(* CODESYS project KotelnayLesnay.project
   Title: KotelnayLesnay
   Author: User
   Version: 0.0.0.178

Project tree, tasks and I/O mapping:
  MyController : TM241CE40T/U, Schneider Electric, order no. TM241CE40T/U, version 4.0.6.18
    application Application
      libraries: Toolbox_Advance, 1.0.1.0 (Schneider Electric); Toolbox, 2.2.0.0 (Schneider Electric); SysTimeRtc, 3.5.1.0 (System)
      task MAST (cyclic, interval 20 ms, priority 15, watchdog 100 ms x 1) calls INPUT, AnalogSensers, PidMeteoVlv, PidGvs, ManualMode, year_month_day, DQ
      global variables GVL
      program INPUT [ST]
      program DQ [ST]
      program ManualMode [LD]
      program AnalogSensers [FBD]
      global variables GVL_RETAIN
      program PidMeteoVlv [FBD]
      function block OutputLimit [ST]
      program year_month_day [CFC]
      function block SendData [CFC]
      function CRC16 [ST]
      function block CRC_16 [ST]
      function block array_to_float [ST]
      data type word_real
      program PidGvs [FBD]
      function block InitializationTmpGrafik [ST]
    A1DI : Digital Inputs, Schneider Electric, version 4.0.6.18
        input  idwDI_IDW0 : DWORD  // IDW0
        input  X0 : BOOL  // IDW0.I0
        input  X1 : BOOL  // IDW0.I1
        input  X2 : BOOL  // IDW0.I2
        input  X3 : BOOL  // IDW0.I3
        input  X4 : BOOL  // IDW0.I4
        input  X5 : BOOL  // IDW0.I5
        input  X6 : BOOL  // IDW0.I6
        input  X7 : BOOL  // IDW0.I7
        input  X8 : BOOL  // IDW0.I8
        input  X9 : BOOL  // IDW0.I9
        input  X10 : BOOL  // IDW0.I10
        input  X11 : BOOL  // IDW0.I11
        input  X12 : BOOL  // IDW0.I12
        input  X13 : BOOL  // IDW0.I13
        input  X14 : BOOL  // IDW0.I14
        input  X15 : BOOL  // IDW0.I15
        input  X16 : BOOL  // IDW0.I16
        input  X17 : BOOL  // IDW0.I17
        input  X18 : BOOL  // IDW0.I18
        input  X19 : BOOL  // IDW0.I19
        input  X20 : BOOL  // IDW0.I20
        input  X21 : BOOL  // IDW0.I21
        input  X22 : BOOL  // IDW0.I22
        input  X23 : BOOL  // IDW0.I23
        input  ibDI_IB1 : BYTE  // IB1
    A1DQ : Digital Outputs, Schneider Electric, version 4.0.6.18
        output Y0 : BOOL  // QW0.Q0
        output Y1 : BOOL  // QW0.Q1
        output Y2 : BOOL  // QW0.Q2
        output Y3 : BOOL  // QW0.Q3
        output Y4 : BOOL  // QW0.Q4
        output Y5 : BOOL  // QW0.Q5
        output Y6 : BOOL  // QW0.Q6
        output Y7 : BOOL  // QW0.Q7
        output Y8 : BOOL  // QW0.Q8
        output Y9 : BOOL  // QW0.Q9
        output Y10 : BOOL  // QW0.Q10
        output Y11 : BOOL  // QW0.Q11
        output Y12 : BOOL  // QW0.Q12
        output Y13 : BOOL  // QW0.Q13
        output Y14 : BOOL  // QW0.Q14
        output Y15 : BOOL  // QW0.Q15
        output qbDQ_QB1 : BYTE  // QB1
        unmapped channels: QW0
    Counters : Counters, Schneider Electric, version 4.0.6.18
    Pulse_Generators : Pulse Generators, Schneider Electric, version 4.0.6.18
    Cartridge_1 : Cartridge, Schneider Electric, version 4.0.6.18
    Cartridge_2 : Cartridge, Schneider Electric, version 4.0.6.18
    IO_Bus : IO bus - TM3, Schneider Electric, version 4.0.6.18
      A12DI : TM3DI32K, Schneider Electric, order no. TM3DI32K, version 1.0.1.3
          input  idwModule_2_ID0 : DWORD  // ID0
          input  _1X0 : BOOL  // ID0.I0
          input  _1X1 : BOOL  // ID0.I1
          input  _1X2 : BOOL  // ID0.I2
          input  _1X3 : BOOL  // ID0.I3
          input  _1X4 : BOOL  // ID0.I4
          input  _1X5 : BOOL  // ID0.I5
          input  _1X6 : BOOL  // ID0.I6
          input  _1X7 : BOOL  // ID0.I7
          input  _1X8 : BOOL  // ID0.I8
          input  _1X9 : BOOL  // ID0.I9
          input  _1X10 : BOOL  // ID0.I10
          input  _1X11 : BOOL  // ID0.I11
          input  _1X12 : BOOL  // ID0.I12
          input  _1X13 : BOOL  // ID0.I13
          input  _1X14 : BOOL  // ID0.I14
          input  _1X15 : BOOL  // ID0.I15
          input  _1X16 : BOOL  // ID0.I16
          input  _1X17 : BOOL  // ID0.I17
          input  _1X18 : BOOL  // ID0.I18
          input  _1X19 : BOOL  // ID0.I19
          input  _1X24 : BOOL  // ID0.I24
          input  _1X25 : BOOL  // ID0.I25
          input  _1X23 : BOOL  // ID0.I27
          input  _1X20 : BOOL  // ID0.I28
          input  _1X21 : BOOL  // ID0.I29
          input  _1X22 : BOOL  // ID0.I30
      A13AI : TM3AI8/G, Schneider Electric, order no. TM3AI8/G, version 1.0.0.17
          settings: KPI Configuration.KPI Configuration[0] = 35; KPI Configuration.KPI Configuration[1] = 35; KPI Configuration.KPI Configuration[2] = 35; KPI Configuration.KPI Configuration[3] = 35; KPI Configuration.KPI Configuration[4] = 35; KPI Configuration.KPI Configuration[8] = 160; KPI Configuration.KPI Configuration[9] = 15; KPI Configuration.KPI Configuration[10] = 160; KPI Configuration.KPI Configuration[11] = 15; KPI Configuration.KPI Configuration[12] = 160; KPI Configuration.KPI Configuration[13] = 15; KPI Configuration.KPI Configuration[14] = 160; KPI Configuration.KPI Configuration[15] = 15; KPI Configuration.KPI Configuration[16] = 160; KPI Configuration.KPI Configuration[17] = 15; KPI Configuration.KPI Configuration[24] = 32; KPI Configuration.KPI Configuration[25] = 78; KPI Configuration.KPI Configuration[26] = 32; KPI Configuration.KPI Configuration[27] = 78; KPI Configuration.KPI Configuration[28] = 32; KPI Configuration.KPI Configuration[29] = 78; KPI Configuration.KPI Configuration[30] = 32; KPI Configuration.KPI Configuration[31] = 78; KPI Configuration.KPI Configuration[32] = 32; KPI Configuration.KPI Configuration[33] = 78; KPI Configuration.KPI Configuration[40] = 10; KPI Configuration.KPI Configuration[42] = 10; KPI Configuration.KPI Configuration[44] = 10; KPI Configuration.KPI Configuration[46] = 10; KPI Configuration.KPI Configuration[48] = 10
          input  PT3 : INT  // IW0
          input  PT4 : INT  // IW1
          input  PT6 : INT  // IW2
          input  PT5 : INT  // IW3
          input  PT8 : INT  // IW4
          input  PT10 : INT  // IW5
          input  iiModule_3_IW6 : INT  // IW6
          input  iiModule_3_IW7 : INT  // IW7
          input  ibModule_3_IBStatusIW0 : BYTE  // IBStatusIW0
          input  ibModule_3_IBStatusIW1 : BYTE  // IBStatusIW1
          input  ibModule_3_IBStatusIW2 : BYTE  // IBStatusIW2
          input  ibModule_3_IBStatusIW3 : BYTE  // IBStatusIW3
          input  ibModule_3_IBStatusIW4 : BYTE  // IBStatusIW4
          input  ibModule_3_IBStatusIW5 : BYTE  // IBStatusIW5
          input  ibModule_3_IBStatusIW6 : BYTE  // IBStatusIW6
          input  ibModule_3_IBStatusIW7 : BYTE  // IBStatusIW7
      A14AI : TM3TI4/G, Schneider Electric, order no. TM3TI4/G, version 1.0.1.5
          settings: KPI Configuration.KPI Configuration[0] = 77; KPI Configuration.KPI Configuration[1] = 77; KPI Configuration.KPI Configuration[2] = 77; KPI Configuration.KPI Configuration[3] = 77; KPI Configuration.KPI Configuration[4] = 48; KPI Configuration.KPI Configuration[5] = 248; KPI Configuration.KPI Configuration[6] = 48; KPI Configuration.KPI Configuration[7] = 248; KPI Configuration.KPI Configuration[8] = 48; KPI Configuration.KPI Configuration[9] = 248; KPI Configuration.KPI Configuration[10] = 48; KPI Configuration.KPI Configuration[11] = 248; KPI Configuration.KPI Configuration[12] = 52; KPI Configuration.KPI Configuration[13] = 33; KPI Configuration.KPI Configuration[14] = 52; KPI Configuration.KPI Configuration[15] = 33; KPI Configuration.KPI Configuration[16] = 52; KPI Configuration.KPI Configuration[17] = 33; KPI Configuration.KPI Configuration[18] = 52; KPI Configuration.KPI Configuration[19] = 33
          input  TE1 : INT  // IW0
          input  TE2 : INT  // IW1
          input  TE3 : INT  // IW2
          input  TE4 : INT  // IW3
          input  ibModule_4_IBStatusIW0 : BYTE  // IBStatusIW0
          input  ibModule_4_IBStatusIW1 : BYTE  // IBStatusIW1
          input  ibModule_4_IBStatusIW2 : BYTE  // IBStatusIW2
          input  ibModule_4_IBStatusIW3 : BYTE  // IBStatusIW3
      A15AI : TM3TI4/G, Schneider Electric, order no. TM3TI4/G, version 1.0.1.5
          settings: KPI Configuration.KPI Configuration[0] = 77; KPI Configuration.KPI Configuration[1] = 77; KPI Configuration.KPI Configuration[2] = 77; KPI Configuration.KPI Configuration[3] = 77; KPI Configuration.KPI Configuration[4] = 48; KPI Configuration.KPI Configuration[5] = 248; KPI Configuration.KPI Configuration[6] = 48; KPI Configuration.KPI Configuration[7] = 248; KPI Configuration.KPI Configuration[8] = 48; KPI Configuration.KPI Configuration[9] = 248; KPI Configuration.KPI Configuration[10] = 48; KPI Configuration.KPI Configuration[11] = 248; KPI Configuration.KPI Configuration[12] = 52; KPI Configuration.KPI Configuration[13] = 33; KPI Configuration.KPI Configuration[14] = 52; KPI Configuration.KPI Configuration[15] = 33; KPI Configuration.KPI Configuration[16] = 52; KPI Configuration.KPI Configuration[17] = 33; KPI Configuration.KPI Configuration[18] = 52; KPI Configuration.KPI Configuration[19] = 33
          input  TE5 : INT  // IW0
          input  TE6 : INT  // IW1
          input  TE7 : INT  // IW2
          input  TE8 : INT  // IW3
          input  ibModule_5_IBStatusIW0 : BYTE  // IBStatusIW0
          input  ibModule_5_IBStatusIW1 : BYTE  // IBStatusIW1
          input  ibModule_5_IBStatusIW2 : BYTE  // IBStatusIW2
          input  ibModule_5_IBStatusIW3 : BYTE  // IBStatusIW3
      A16AI : TM3TI4/G, Schneider Electric, order no. TM3TI4/G, version 1.0.1.5
          settings: KPI Configuration.KPI Configuration[0] = 77; KPI Configuration.KPI Configuration[4] = 48; KPI Configuration.KPI Configuration[5] = 248; KPI Configuration.KPI Configuration[12] = 52; KPI Configuration.KPI Configuration[13] = 33
          input  TE9 : INT  // IW0
          input  iiModule_6_IW1 : INT  // IW1
          input  iiModule_6_IW2 : INT  // IW2
          input  iiModule_6_IW3 : INT  // IW3
          input  ibModule_6_IBStatusIW0 : BYTE  // IBStatusIW0
          input  ibModule_6_IBStatusIW1 : BYTE  // IBStatusIW1
          input  ibModule_6_IBStatusIW2 : BYTE  // IBStatusIW2
          input  ibModule_6_IBStatusIW3 : BYTE  // IBStatusIW3
      A11DQ : TM3DQ32TK, Schneider Electric, order no. TM3DQ32TK, version 1.0.1.3
          output _1Y0 : BOOL  // QD0.Q0
          output _1Y1 : BOOL  // QD0.Q1
          output _1Y2 : BOOL  // QD0.Q2
          output _1Y3 : BOOL  // QD0.Q3
          output _1Y4 : BOOL  // QD0.Q4
          unmapped channels: QD0
    COM_Bus : COM bus, Schneider Electric, version 4.0.6.18
    Ethernet_1 : Ethernet Network, Schneider Electric, version 4.0.6.18
        settings: IPAddress = [192, 168, 0, 2]; SubnetMask = [255, 255, 255, 0]; GatewayAddress = [192, 168, 0, 1]; WebServer = TRUE; FTP Server = TRUE; SoMachine Protocol = TRUE; Modbus Server = TRUE; NetManage Protocol = TRUE; SNMP protocol = TRUE; Enable Routing = FALSE; WebVisu protocol = TRUE; DHCP Server Active = TRUE
    Serial_Line_1 : Serial line, Schneider Electric, version 4.0.6.18
      SoMachine_Network_Manager : SoMachine-Network Manager, Schneider Electric, version 4.0.0.2
    Serial_Line_2 : Serial line, Schneider Electric, version 4.0.6.18
      Modbus_IOScanner : Modbus IOScanner, Schneider Electric, version 3.5.3.8
          settings: Transmission = 'RTU'; ResponseTimeout = 1000; TimeBetweenFrames = 1000
        Boiler_2 : Generic Modbus Slave, Schneider Electric, version 3.5.3.9
            settings: SlaveAddress = 32; ResponseTimeout = 1000; Read_7_tags.Function Code = 3; Read_7_tags.Read Offset = 16#0000; Read_7_tags.Read Length = 8; Read_7_tags.Write Offset = 0; Read_7_tags.Write Length = 0; Read_7_tags.Cycle Time = 1000; Start_Stop.Function Code = 6; Start_Stop.Read Offset = 0; Start_Stop.Read Length = 0; Start_Stop.Write Offset = 16#0080; Start_Stop.Write Length = 1; Start_Stop.Cycle Time = 1000; Ustavka_TMP_CO_2.Function Code = 6; Ustavka_TMP_CO_2.Read Offset = 0; Ustavka_TMP_CO_2.Read Length = 0; Ustavka_TMP_CO_2.Write Offset = 16#0081; Ustavka_TMP_CO_2.Write Length = 1; Ustavka_TMP_CO_2.Cycle Time = 1000; StartStopStait.Function Code = 3; StartStopStait.Read Offset = 16#0080; StartStopStait.Read Length = 1; StartStopStait.Write Offset = 0; StartStopStait.Write Length = 0; StartStopStait.Cycle Time = 1000
            input  Application.StaitBoiler2 : WORD  // Read_7_tags.Read_7_tags[0]
            input  Application.TmpCoBoiler2 : WORD  // Read_7_tags.Read_7_tags[1]
            input  Application.TmpRecirculationBoiler2 : WORD  // Read_7_tags.Read_7_tags[2]
            input  Application.TmpFire1_Boiler2 : WORD  // Read_7_tags.Read_7_tags[3]
            input  Application.TmpFire2_Boiler2 : WORD  // Read_7_tags.Read_7_tags[4]
            input  Application.TmpShnek1_Boiler2 : WORD  // Read_7_tags.Read_7_tags[5]
            input  Application.TmpShnek2_Boiler2 : WORD  // Read_7_tags.Read_7_tags[6]
            input  Application.ErrBoiler2 : WORD  // Read_7_tags.Read_7_tags[7]
            output Application._START_STOP_BOILER2 : ARRAY[0..0] OF WORD  // Start_Stop
            output Application._USTAVKA_TMP_CO_2 : ARRAY[0..0] OF WORD  // Ustavka_TMP_CO_2
            input  Application.StartStopStait2 : ARRAY[0..0] OF WORD  // StartStopStait
            unmapped channels: Read_7_tags
        GVS : Generic Modbus Slave, Schneider Electric, version 3.5.3.9
            settings: SlaveAddress = 4; ResponseTimeout = 1000; KP.Function Code = 6; KP.Read Offset = 0; KP.Read Length = 0; KP.Write Offset = 16#0FBF; KP.Write Length = 1; KP.Cycle Time = 1000; KI.Function Code = 6; KI.Read Offset = 0; KI.Read Length = 0; KI.Write Offset = 16#0FC0; KI.Write Length = 1; KI.Cycle Time = 1000; KD.Function Code = 6; KD.Read Offset = 0; KD.Read Length = 0; KD.Write Offset = 16#0FC1; KD.Write Length = 1; KD.Cycle Time = 1000; CURRENT.Function Code = 3; CURRENT.Read Offset = 16#006A; CURRENT.Read Length = 1; CURRENT.Write Offset = 0; CURRENT.Write Length = 0; CURRENT.Cycle Time = 1000; FREQUENSY.Function Code = 3; FREQUENSY.Read Offset = 16#0069; FREQUENSY.Read Length = 1; FREQUENSY.Write Offset = 0; FREQUENSY.Write Length = 0; FREQUENSY.Cycle Time = 1000; SET_POINT.Function Code = 6; SET_POINT.Read Offset = 0; SET_POINT.Read Length = 0; SET_POINT.Write Offset = 16#0006; SET_POINT.Write Length = 1; SET_POINT.Cycle Time = 1000
            output Application._KP_GVS : ARRAY[0..0] OF WORD  // KP
            output Application._KI_GVS : ARRAY[0..0] OF WORD  // KI
            output Application._KD_GVS : ARRAY[0..0] OF WORD  // KD
            input  Application._CURRENT_GVS : ARRAY[0..0] OF WORD  // CURRENT
            input  Application._FREQUENSY_GVS : ARRAY[0..0] OF WORD  // FREQUENSY
            output Application._SET_POINT_GVS : ARRAY[0..0] OF WORD  // SET_POINT
        NETWORK_1 : Generic Modbus Slave, Schneider Electric, version 3.5.3.9
            settings: SlaveAddress = 2; ResponseTimeout = 1000; KP.Function Code = 6; KP.Read Offset = 0; KP.Read Length = 0; KP.Write Offset = 16#0FBF; KP.Write Length = 1; KP.Cycle Time = 1000; KI.Function Code = 6; KI.Read Offset = 0; KI.Read Length = 0; KI.Write Offset = 16#0FC0; KI.Write Length = 1; KI.Cycle Time = 1000; KD.Function Code = 6; KD.Read Offset = 0; KD.Read Length = 0; KD.Write Offset = 16#0FC1; KD.Write Length = 1; KD.Cycle Time = 1000; CURRENT.Function Code = 3; CURRENT.Read Offset = 16#006A; CURRENT.Read Length = 1; CURRENT.Write Offset = 0; CURRENT.Write Length = 0; CURRENT.Cycle Time = 1000; FREQUENSY.Function Code = 3; FREQUENSY.Read Offset = 16#0069; FREQUENSY.Read Length = 1; FREQUENSY.Write Offset = 0; FREQUENSY.Write Length = 0; FREQUENSY.Cycle Time = 1000; SET_POINT.Function Code = 6; SET_POINT.Read Offset = 0; SET_POINT.Read Length = 0; SET_POINT.Write Offset = 16#0006; SET_POINT.Write Length = 1; SET_POINT.Cycle Time = 1000
            output Application._KP_NETWORK_1 : ARRAY[0..0] OF WORD  // KP
            output Application._KI_NETWORK_1 : ARRAY[0..0] OF WORD  // KI
            output Application._KD_NETWORK_1 : ARRAY[0..0] OF WORD  // KD
            input  Application._CURRENT_NETWORK_1 : ARRAY[0..0] OF WORD  // CURRENT
            input  Application._FREQUENSY_NETWORK_1 : ARRAY[0..0] OF WORD  // FREQUENSY
            output Application._SET_POINT_NETWORK_1 : ARRAY[0..0] OF WORD  // SET_POINT
        NETWORK_2 : Generic Modbus Slave, Schneider Electric, version 3.5.3.9
            settings: SlaveAddress = 3; ResponseTimeout = 1000; KP.Function Code = 6; KP.Read Offset = 0; KP.Read Length = 0; KP.Write Offset = 16#0FBF; KP.Write Length = 1; KP.Cycle Time = 1000; KI.Function Code = 6; KI.Read Offset = 0; KI.Read Length = 0; KI.Write Offset = 16#0FC0; KI.Write Length = 1; KI.Cycle Time = 1000; KD.Function Code = 6; KD.Read Offset = 0; KD.Read Length = 0; KD.Write Offset = 16#0FC1; KD.Write Length = 1; KD.Cycle Time = 1000; CURRENT.Function Code = 3; CURRENT.Read Offset = 16#006A; CURRENT.Read Length = 1; CURRENT.Write Offset = 0; CURRENT.Write Length = 0; CURRENT.Cycle Time = 1000; FREQUENSY.Function Code = 3; FREQUENSY.Read Offset = 16#0069; FREQUENSY.Read Length = 1; FREQUENSY.Write Offset = 0; FREQUENSY.Write Length = 0; FREQUENSY.Cycle Time = 1000; SET_POINT.Function Code = 6; SET_POINT.Read Offset = 0; SET_POINT.Read Length = 0; SET_POINT.Write Offset = 16#0006; SET_POINT.Write Length = 1; SET_POINT.Cycle Time = 1000
            output Application._KP_NETWORK_2 : ARRAY[0..0] OF WORD  // KP
            output Application._KI_NETWORK_2 : ARRAY[0..0] OF WORD  // KI
            output Application._KD_NETWORK_2 : ARRAY[0..0] OF WORD  // KD
            input  Application._CURRENT_NETWORK_2 : ARRAY[0..0] OF WORD  // CURRENT
            input  Application._FREQUENSY_NETWORK_2 : ARRAY[0..0] OF WORD  // FREQUENSY
            output Application._SET_POINT_NETWORK_2 : ARRAY[0..0] OF WORD  // SET_POINT
        Boiler_1 : Generic Modbus Slave, Schneider Electric, version 3.5.3.9
            settings: SlaveAddress = 33; ResponseTimeout = 1000; Ustavka_TMP_CO_1.Function Code = 6; Ustavka_TMP_CO_1.Read Offset = 0; Ustavka_TMP_CO_1.Read Length = 0; Ustavka_TMP_CO_1.Write Offset = 16#0081; Ustavka_TMP_CO_1.Write Length = 1; Ustavka_TMP_CO_1.Cycle Time = 1000; StartStopStait.Function Code = 3; StartStopStait.Read Offset = 16#0080; StartStopStait.Read Length = 1; StartStopStait.Write Offset = 0; StartStopStait.Write Length = 0; StartStopStait.Cycle Time = 1000; Read_7_regs.Function Code = 3; Read_7_regs.Read Offset = 16#0000; Read_7_regs.Read Length = 8; Read_7_regs.Write Offset = 0; Read_7_regs.Write Length = 0; Read_7_regs.Cycle Time = 1000; Start_stop.Function Code = 6; Start_stop.Read Offset = 0; Start_stop.Read Length = 0; Start_stop.Write Offset = 16#0080; Start_stop.Write Length = 1; Start_stop.Cycle Time = 1000
            output Application._USTAVKA_TMP_CO_1 : ARRAY[0..0] OF WORD  // Ustavka_TMP_CO_1
            input  Application.StartStopStait1 : WORD  // StartStopStait.StartStopStait[0]
            input  Application.StaitBoiler1 : WORD  // Read_7_regs.Read_7_regs[0]
            input  Application.TmpCoBoiler1 : WORD  // Read_7_regs.Read_7_regs[1]
            input  Application.TmpRecirculationBoiler1 : WORD  // Read_7_regs.Read_7_regs[2]
            input  Application.TmpFire1_Boiler1 : WORD  // Read_7_regs.Read_7_regs[3]
            input  Application.TmpFire2_Boiler1 : WORD  // Read_7_regs.Read_7_regs[4]
            input  Application.TmpShnek1_Boiler1 : WORD  // Read_7_regs.Read_7_regs[5]
            input  Application.TmpShnek2_Boiler1 : WORD  // Read_7_regs.Read_7_regs[6]
            input  Application.ErrBoiler1 : WORD  // Read_7_regs.Read_7_regs[7]
            output Application._START_STOP_BOILER1 : ARRAY[0..0] OF WORD  // Start_stop
            unmapped channels: StartStopStait, Read_7_regs
*)

// MyController/Application/word_real
TYPE word_real :
UNION
	realValue:REAL;
	awModbusByte: ARRAY[1..4] OF BYTE;
END_UNION
END_TYPE

// MyController/Application/GVL
VAR_GLOBAL
	//--------------------------------------------------------
	//--------A1----------------------------------------------
	//--------------------------------------------------------
	
	VlvGass AT %MX2.10: BOOL;// Газовый клапан
	Gassed AT %MX2.11: BOOL;// Загазованность
	VlvDranchOpen AT %MX2.12: BOOL;// Открытие клапана дренчера
	PressInLoadGvs_K14 AT %MX2.13: BOOL;// Давление во всасывающем трубопроводе насосов загрузочных теплообменников ГВС К14
	MonitorFlwWtrBoiler1 AT %MX2.14: BOOL;// Контроль расхода воды через котел 1
	PmpRcr1InAutoMode AT %MX2.15: BOOL;// Насос рециркуляции 1 в авторежиме
	
	PmpRcr2InAutoMode AT %MX58.0: BOOL;// Насос рециркуляции 2 в авторежиме
	PmpRcr3InAutoMode AT %MX58.1: BOOL;// Насос рециркуляции 3 в авторежиме
	PmpWtr1InAutoMode AT %MX58.2: BOOL;// Насос исходной воды 1 в авторежиме
	PmpWtr2InAutoMode AT %MX58.3: BOOL;// Насос исходной воды 2 в авторежиме
	PmpRcr1On AT %MX58.4: BOOL;// Насос рециркуляции 1 включен
	PmpRcr2On AT %MX58.5: BOOL;// Насос рециркуляции 2 включен
	PmpRcr3On AT %MX58.6: BOOL;// Насос рециркуляции 3 включен
	PmpWtr1On AT %MX58.7: BOOL;// Насос исходной воды 1 включен
	PmpWtr2On AT %MX58.8: BOOL;// Насос исходной воды 2 включен
	MonitorFlwWtrBoiler2 AT %MX58.9: BOOL;// Контроль расхода воды через котел 2
	PmpsGvsInAtoMode AT %MX58.10: BOOL;// Насосы сетевые ГВС 1 и 2 в авторежиме
	PmpGvs1FromPch AT %MX58.11: BOOL;// Насос сетевой ГВС 1 работа от ПЧ
	PmpGvs2FromPch AT %MX58.12: BOOL;// Насос сетевой ГВС 2 работа от ПЧ
	WorkPchGvs1_2 AT %MX58.13: BOOL;// Работ ПЧ сетевых насосов ГВС 1, 2 
	ErrPchNetPumpsGvs1_2 AT %MX58.14: BOOL;// Авария ПЧ сетевых насосов ГВС 1, 2
	PmpNet1_2InAutoMode AT %MX58.15: BOOL;// Насовы сетевые 1, 2 в авто режиме
	FanInAutoMode AT %MX60.0: BOOL;// Вентилятор вытяжной в авто режиме
	PmpsLoadGvsInAutoMode AT %MX60.1: BOOL;// Насосы загрузочные ГВС 1, 2 в авторежиме
	PmpNet1On AT %MX60.2: BOOL;// Насос тетевой 1 запущен
	//--------------------------------------------------------
	//-------A1-----------------------------------------------
	//--------------------------------------------------------
	Rezerv: BOOL;
	RunAlarm: BOOL;// включить аварию
	RunSiren: BOOL;// включить сирену
	RunPmpRcr1: BOOL;// запустить насос рециркуляции 1
	RunPmpRcr2: BOOL;// запустить насос рециркуляции 2
	RunPmpRcr3: BOOL;// запустить насос рециркуляции 3
	RunPmpWtr1: BOOL;// запустить насос исходной воды 1
	RunPmpWtr2: BOOL;// запустить насос исходной воды 2
	RumPmpGvs1FromPch: BOOL;// запустить насос сетевой ГВС 1 от ПЧ
	RumPmpGvs2FromPch: BOOL;// запустить насос сетевой ГВС 2 от ПЧ
	StartPchGvs1_2: BOOL;// старт насосов сетевых от ПЧ
	RunPmpNet1: BOOL;// запустить насос сетевой воды 1
	RunPmpNet2: BOOL;// запустить насос сетевой воды 2
	RunFan: BOOL;// запустить вытяжной вентилятор
	RunPmpLoadGvs1: BOOL;// запустить насос 1 загрузги ГВС 
	RunPmpLoadGvs2: BOOL;// запустить насос 2 загрузги ГВС
	//--------------------------------------------------------
	//--------A1.1--------------------------------------------
	//--------------------------------------------------------		
	RunVlvDrench: BOOL;// включить клапан дренчерной завесы
	RunOpnMeteoVlv: BOOL;// открыть погодозависимый клапан
	RunClsMeteoVlv: BOOL;// закрыть погодозависимый клапан
	RunOpnVlvLoadGvs: BOOL;// открыть клапан загрузки ГВС
	RunClsVlvLoadGvs: BOOL;// закрыть клапан загрузки ГВС
	//--------------------------------------------------------
	//-----A1.2-----------------------------------------------
	//--------------------------------------------------------
	PmpNet2On AT %MX60.3: BOOL;// Насос сетевой 2 запущен
	FanOn AT %MX60.4: BOOL;// Вытяжной вентилятор запущен
	PmpLoadGvs1On AT %MX60.5: BOOL;// Насос загрузочный ГВС 1 включен
	PmpLoadGvs2On AT %MX60.6: BOOL;// Насос загрузочный ГВС 2 включен
	WorkPchPmpNet1 AT %MX60.7: BOOL;// Работа ПЧ насоса сетевого 1
	ErrPchPmpNet1 AT %MX60.8: BOOL;// Авария ПЧ насоса сетевого 1
	WorkPchPmpNet2 AT %MX60.9: BOOL;// Работа ПЧ сетевого насоса 2
	ErrPchPmpNet2 AT %MX60.10: BOOL;// Авария ПЧ сетевого насоса 2
	MtrMeteoInAutoMode AT %MX60.11: BOOL;// Электропривод на погодное регулинование в авторежиме
	MtrLoadGvsInAutoMode AT %MX60.12: BOOL;// Электропривод загрузки теплообменника ГВС в авторежиме
	PressOut1_K2 AT %MX60.13: BOOL;// Давление в напорном трубопроводе котлового насоса К2 №1
	PressIn1_K2 AT %MX60.14: BOOL;// Давление во всасывающем трубопроводе котлового насоса К2 №1
	PressOut2_K2 AT %MX60.15: BOOL;// Давление в напорном трубопроводе котлового насоса К2 №2
	PressIn2_K2 AT %MX62.0: BOOL;// Давление во всасывающем трубопроводе котлового насоса К2 №2
	PressOut3_K7 AT %MX62.1: BOOL;// Давление в напорном трубопроводе котлового насоса К7 №3
	PressIn3_K7 AT %MX62.2: BOOL;// Давление во всасывающем трубопроводе котлового насоса К7 №3
	PressNet_K3 AT %MX62.3: BOOL;// Давление в общем напорном трубопроводе сетевых насосов К3
	PressInNet_K5 AT %MX62.4: BOOL;// Давление в общем всасывающем трубопроводе сетевых насосов К5
	PressOutGvs_K6 AT %MX62.5: BOOL;// Давление в общем напорном трубопроводе сетевых насосов ГВС К6
	PressInGvs_K5 AT %MX62.6: BOOL;// Давление в общем всасывающем трубопроводе сетевых насосов ГВС К5
	PressOutWtr_K4 AT %MX62.7: BOOL;// Давление в общем напорном трубопроводе насосов исходной воды К4
	PressInWtr_K4 AT %MX62.8: BOOL;// Давление в общем всасывающем трубопроводе насосов исходной воды К4
	PresBefoWtrPrepar1 AT %MX62.9: BOOL;// Давление перед водоподготовкой NC контакт
	PresBefoWtrPrepar2 AT %MX62.10: BOOL;// Давление перед водоподготовкой NO контакт
	PressOutLoadGvs_K14 AT %MX62.11: BOOL;// Давление в общем напорном трубопроводе насосов загрузочных теплообменников ГВС К14
	HandMode AT %MX62.12: BOOL;
	StartStopBoiler AT %MX62.13: BOOL;
	BtnOnOffSiren AT %MX62.14: BOOL;// Кнопка отключения сирены
	WorkOnTask AT %MX62.15: BOOL;// Работать по уставке
	
	//--------------------------------------------------------
	//-----A1.3-----------------------------------------------
	//--------------------------------------------------------
	PressPodachi AT %MW3: INT;// Давление в прямом сетевом трубопроводе на выходе из котельной РТ3
	PressObratki AT %MW4: INT;// Давление в обратно сетевом трубопроводе после фильтра РТ4
	PressPodachiGvs AT %MW5: INT;// Давление в прямом трубопроводе ГВС на выходе из котельной РТ6
	PressObratkiGvs AT %MW6: INT;// Давление в обратном трубопроводе ГВС на входе в котельную РТ5
	PressWtr AT %MW7: INT;// Давление на вводе холодной воды РТ8
	PressGass AT %MW16: INT;// Давление газа на вводе в котельную РТ10
	//--------------------------------------------------------
	//-----A1.4-----------------------------------------------
	//--------------------------------------------------------
	TmpWtrInBoilerK8 AT %MW8: INT;// Температура воды на входе в котел К8 (ТЕ1)
	TmpWtrIn1BoilerK2 AT %MW9: INT;// Температура воды на входе в котел К2 №1(ТЕ2)
	TmpWtrIn2BoilerK2 AT %MW10: INT;// Температура воды на входе в котел К2 №2(ТЕ3)
	TmpWtrPodachi AT %MW11: INT;// Температура воды в прямом сетевом трубопроводе на выходе из котельной (ТЕ4)
	//--------------------------------------------------------
	//-----A1.5-----------------------------------------------
	//--------------------------------------------------------
	TmpWtrObratki AT %MW12: INT;// Температура воды в обратном сетевом трубопроводе на входе в котельную (ТЕ5)
	TmpWtrPodachiGvs AT %MW13: INT;// Температура воды в прямом сетевом трубопроводе ГВС на выходе из котельной (ТЕ6)
	TmpWtrObratkiGvs AT %MW14: INT;// Температура воды в обратном сетевом трубопроводе ГВС на входе в котельную (ТЕ7)
	TmpAir AT %MW15: INT;// Температура наружнего воздуха
	//--------------------------------------------------------
	//-----A1.6-----------------------------------------------
	//--------------------------------------------------------
	TmpWtrGvs AT %MW2: INT;// Температура воды в трубопроводе ГВС на входе из теплообменников ГВС(ТЕ8)
	//--------------------------------------------------------
	//-----ManualMode-----------------------------------------	
	//--------------------------------------------------------
	BtnRunAlarm AT %MX0.0: BOOL;// Кнопка включить аварию
	BtnRunSiren AT %MX0.1: BOOL;// Кнопка включить сирену	
	BtnRunPmpRcr1 AT %MX0.2: BOOL;// Кнопка запустить насос рециркуляции 1	
	BtnRunPmpRcr2 AT %MX0.3: BOOL;// Кнопка запустить насос рециркуляции 2	
	BtnRunPmpRcr3 AT %MX0.4: BOOL;// Кнопка запустить насос рециркуляции 3	
	BtnRunPmpWtr1 AT %MX0.5: BOOL;// Кнопка запустить насос исходной воды 1	
	BtnRunPmpWtr2 AT %MX0.6: BOOL;// Кнопка запустить насос исходной воды 2	
	BtnRumPmpGvs1FromPch AT %MX0.7: BOOL;// Кнопка запустить насос сетевой 1 ГВС от ПЧ	
	BtnRumPmpGvs2FromPch AT %MX0.8: BOOL;// Кнопка запустить насос сетевой 2 ГВС от ПЧ	
	BtnStartPchGvs1_2 AT %MX0.9: BOOL;// Кнопка старт насосов сетевых 1,2 от ПЧ	(включить ПЧ)
	BtnRumPmpNet1 AT %MX0.10: BOOL;// Кнопка запустить насос сетевой воды 1	
	BtnRumPmpNet2 AT %MX0.11: BOOL;// Кнопка запустить насос сетевой воды 2	
	BtnRunFan AT %MX0.12: BOOL;// Кнопка запустить вытяжной вентилятор	
	BtnRunPmpLoadGvs1 AT %MX0.13: BOOL;// Кнопка запустить насос 1 загрузги ГВС 	
	BtnRunPmpLoadGvs2 AT %MX0.14: BOOL;// Кнопка запустить насос 2 загрузги ГВС	
	BtnRunVlvDrench AT %MX0.15: BOOL;// Кнопка включить клапан дренчерной завесы	
	BtnRunOpnMeteoVlv AT %MX2.0: BOOL;// Кнопка открыть погодозависимый клапан	
	BtnRunClsMeteoVlv AT %MX2.1: BOOL;// Кнопка закрыть погодозависимый клапан	
	BtnRunOpnVlvLoadGvs AT %MX2.2: BOOL;// Кнопка открыть клапан загрузки ГВС
	BtnRunClsVlvLoadGvs AT %MX2.3: BOOL;// Кнопка закрыть клапан загрузки ГВС
	//--------------------------------------------------------
	//-----AnalogSensers-----------------------------------------	
	//--------------------------------------------------------
	ErrPT3 AT %MX2.4: BOOL;
	ErrPT4 AT %mx2.5: BOOL;
	ErrPT5 AT %mx2.6: BOOL;
	ErrPT6 AT %mx2.7: BOOL;
	ErrPT8 AT %mx2.8: BOOL;
	ErrPT10 AT %MX2.9: BOOL;
//-----------Частотники считываем------------
	_KP_GVS: WORD;
	_KI_GVS: WORD;
	_KD_GVS: WORD;
	_CURRENT_GVS: WORD;
	_FREQUENSY_GVS: WORD;
	_SET_POINT_GVS: WORD;
	
	_KP_NETWORK_1: WORD;
	_KI_NETWORK_1: WORD;
	_KD_NETWORK_1: WORD;
	_CURRENT_NETWORK_1: WORD;
	_FREQUENSY_NETWORK_1: WORD;
	_SET_POINT_NETWORK_1: WORD;
		
	_KP_NETWORK_2: WORD;
	_KI_NETWORK_2: WORD;
	_KD_NETWORK_2: WORD;
	_CURRENT_NETWORK_2: WORD;
	_FREQUENSY_NETWORK_2: WORD;
	_SET_POINT_NETWORK_2: WORD;
	

	CURRENT_GVS AT %MW49: WORD;
	FREQUENSY_GVS AT %MW50: WORD;
	

	CURRENT_NETWORK_1 AT %MW55: WORD;
	FREQUENSY_NETWORK_1 AT %MW56: WORD;
		
	CURRENT_NETWORK_2 AT %MW61: WORD;
	FREQUENSY_NETWORK_2 AT %MW62: WORD;
	
	//--------- Котлы-------------------
	//Boiler1: ARRAY[0..7] OF WORD;
	//Boiler2: ARRAY[0..7] OF WORD;
	
	_USTAVKA_TMP_CO_1: INT;
	_START_STOP_BOILER1: WORD;
	StartStopStait1: WORD;
	
	_USTAVKA_TMP_CO_2: INT;
	_START_STOP_BOILER2: WORD;
	StartStopStait2: WORD;
	
	StaitBoiler1: WORD;
	TmpCoBoiler1: WORD;
	TmpRecirculationBoiler1: WORD;
	TmpFire1_Boiler1: WORD;
	TmpFire2_Boiler1: WORD;
	TmpShnek1_Boiler1: WORD;
	TmpShnek2_Boiler1: WORD;	
	ErrBoiler1: WORD;
	
	StaitBoiler2: WORD;
	TmpCoBoiler2: WORD;
	TmpRecirculationBoiler2: WORD;
	TmpFire1_Boiler2: WORD;
	TmpFire2_Boiler2: WORD;
	TmpShnek1_Boiler2: WORD;
	TmpShnek2_Boiler2: WORD;	
	ErrBoiler2: WORD;
	
	//----------------Ручное управление--------------
	HandModeRcr1 AT %MX164.0: BOOL;
	HandModeRcr2 AT %MX164.1: BOOL;
	HandModeRcr3 AT %MX164.2: BOOL;
	HandModeWtr1 AT %MX164.3: BOOL;
	HandModeWtr2 AT %MX164.4: BOOL;
	HandModeNet1 AT %MX164.5: BOOL;
	HandModeNet2 AT %MX164.6: BOOL;
	HandModeGvs AT %MX164.7: BOOL;
	HandModeLoad1 AT %MX164.8: BOOL;
	HandModeLoad2 AT %MX164.9: BOOL;
	HandModeVlvGvs AT %MX164.10: BOOL;
	HandModeMeteo AT %MX164.11: BOOL;
	HandModeBoiler1 AT %MX164.12: BOOL;
	HandModeBoiler2 AT %MX164.13: BOOL;
	
	//----------------Ошибки датчиков--------------
	ErrTE1 AT %MX164.14: BOOL;
	ErrTE2 AT %MX164.15: BOOL;
	
	ErrTE3 AT %MX166.0: BOOL;
	ErrTE4 AT %MX166.1: BOOL;
	ErrTE5 AT %MX166.2: BOOL;
	ErrTE6 AT %MX166.3: BOOL;
	ErrTE7 AT %MX166.4: BOOL;
	ErrTE8 AT %MX166.5: BOOL;
	ErrTE9 AT %MX166.6: BOOL;
	ErrGrafik AT %MX166.7: BOOL;
	ErrAll AT %MX166.8: BOOL;	
	ErrBoiler_1 AT %MX166.9: BOOL;
	ErrBoiler_2 AT %MX166.10: BOOL;
	
	StartStopBoiler_1 AT %MX166.11: BOOL;
	StartStopBoiler_2 AT %MX166.12: BOOL;
	
	//-------------Текущая уставка котла1 и котла2------------
	CurrentUstavka1 AT %MW84: INT;
	CurrentUstavka2 AT %MW85: INT;
	
	//-------------Переменные для уставки времени ПЛК------------	
	uiSetYear AT %MW900: UINT; 
    uiSetMonth AT %MW901: UINT; 
    uiSetDay AT %MW902: UINT; 
    uiSetHour AT %MW903: UINT; 
    uiSetMinute AT %MW904: UINT; 
    uiSetSecond AT %MW905: UINT; 
    uiSetMSecond AT %MW906: UINT;
	
	uiGetYear AT %MW907: UINT; 
    uiGetMonth AT %MW908: UINT; 
    uiGetDay AT %MW909: UINT; 
    uiGetHour AT %MW910: UINT; 
    uiGetMinute AT %MW911: UINT; 
    uiGetSecond AT %MW912: UINT; 
	uiGetDayOfWeek AT %MW913: UINT;
	
	xCommandSetRtc  AT %MX166.13: BOOL;
	xCommandGetRtc  AT %MX166.14: BOOL;
	
	OprosGrands AT %MX166.15: BOOL;
	
	Energy1 AT %MD2000: DWORD;
	Energy2 AT %MD2002: DWORD;
	
END_VAR

// MyController/Application/GVL_RETAIN
VAR_GLOBAL RETAIN
	//--------------------------------------------------------
	//-----AnalogSenser---------------------------------------	
	//--------------------------------------------------------
	PT3_MIN AT %MW17: INT;
	PT3_MAX AT %MW18: INT;
	PT4_MIN AT %MW19: INT;
	PT4_MAX AT %MW20: INT;
	PT5_MIN AT %mw21: INT;
	PT5_MAX AT %mw22: INT;
	PT6_MIN AT %mw23: INT;
	PT6_MAX AT %MW24: INT;
	PT8_MIN AT %MW25: INT;
	PT8_MAX AT %MW26: INT;
	PT10_MIN AT %MW27: INT;
	PT10_MAX AT %MW28: INT;
	//--------------------------------------------------------
	//-----PidMeteoVlv-----------------------------------------	
	//--------------------------------------------------------	
	KpPch AT %MW32: INT;
	TnPch AT %MW33: INT;
	TvPch AT %MW34: INT;
	ManPch AT %MW35: INT;
	MinPch AT %MW36: INT;
	MaxPch AT %MW37: INT;
	ZadaniePch AT %MW38: INT;
	ZadanieVlv AT %MW39: UINT;	
	KpVlv AT %MW40: INT;
	TnVlv AT %MW41: INT;
	TvVlv AT %MW42: INT;
	ManVlv AT %MW43: INT;
	MinVlv AT %MW44: INT;
	MaxVlv AT %MW45: INT;
//-----------Частотники записываем------------	
	KP_GVS AT %MW46: WORD;
	KI_GVS AT %MW47: WORD;
	KD_GVS AT %MW48: WORD;
	SET_POINT_GVS AT %MW51: WORD;
	
	KP_NETWORK_1 AT %MW52: WORD;
	KI_NETWORK_1 AT %MW53: WORD;
	KD_NETWORK_1 AT %MW54: WORD;
	SET_POINT_NETWORK_1 AT %MW57: WORD;
	
	KP_NETWORK_2 AT %MW58: WORD;
	KI_NETWORK_2 AT %MW59: WORD;
	KD_NETWORK_2 AT %MW60: WORD;
	SET_POINT_NETWORK_2 AT %MW63: WORD;
	
	USTAVKA_TMP_CO_1 AT %MW64: INT;
	USTAVKA_TMP_CO_2 AT %MW65: INT;
	

	PositionValve AT %MW86: INT;
	SetPoinGvsVlv AT %MW87: INT;
	ZadanieGvsVlv AT %MW88: INT;	
	KP_GVS_VLV AT %MW89: INT;
	KI_GVS_VLV AT %MW90: INT;
	KD_GVS_VLV AT %MW91: INT;
	MaxGvsVlv AT %MW92: INT;
	PositionGvsValve AT %MW93: INT;
	
	TmpGrafN22 AT %MW94: WORD;
	TmpGrafN19 AT %MW95: WORD;
	TmpGrafN15 AT %MW96: WORD;
	TmpGrafN13 AT %MW97: WORD;
	TmpGrafN10 AT %MW98: WORD;
	TmpGrafN7 AT %MW99: WORD;
	TmpGrafN3 AT %MW100: WORD;
	TmpGraf0 AT %MW101: WORD;
	TmpGraf2 AT %MW102: WORD;
	TmpGraf5 AT %MW103: WORD;
	Tmpgraf10 AT %MW104: WORD;
	
	MinVlvGvs AT %MW105: INT;
	
	KL: ARRAY[0..10] OF POINT;
	
END_VAR

// MyController/Application/INPUT
PROGRAM INPUT
VAR
END_VAR

//------Модуль А1--------------------------------------
VlvGass:=X0;
Gassed:=X1;
VlvDranchOpen:=X2;
MonitorFlwWtrBoiler1:=X3;
PmpRcr1InAutoMode:=X4;
PmpRcr2InAutoMode:=X5;
PmpRcr3InAutoMode:=X6;
PmpWtr1InAutoMode:=X7;
PmpWtr2InAutoMode:=X8;
PmpRcr1On:=X9;
PmpRcr2On:=X10;
PmpRcr3On:=X11;
PmpWtr1On:=X12; 
PmpWtr2On:=X13;
MonitorFlwWtrBoiler2:=X14;
PmpsGvsInAtoMode:=X15;
PmpGvs1FromPch:=X16;
PmpGvs2FromPch:=X17;
WorkPchGvs1_2:=X18;
ErrPchNetPumpsGvs1_2:=X19 AND X15;
PmpNet1_2InAutoMode:=X20;
FanInAutoMode:=X21;
PmpsLoadGvsInAutoMode:=X22;
PmpNet1On:=X23;
//------Модуль А1.2--------------------------------
PmpNet2On:=_1X0;
FanOn:=_1X1;
PmpLoadGvs1On:=_1X2;
PmpLoadGvs2On:=_1X3;
WorkPchPmpNet1:=_1X4;
ErrPchPmpNet1:=_1X5 AND X20;
WorkPchPmpNet2:=_1X6;
ErrPchPmpNet2:=_1X7 AND X20;
MtrMeteoInAutoMode:=_1X8;
MtrLoadGvsInAutoMode:=_1X9;
PressOut1_K2:=NOT _1X10;
PressIn1_K2:=NOT _1X11;
PressOut2_K2:=NOT _1X12;
PressIn2_K2:=NOT _1X13;
PressOut3_K7:=NOT _1X14;
PressIn3_K7:=_1X15;
PressNet_K3:=NOT _1X16;
PressInNet_K5:=NOT _1X17;
PressOutGvs_K6:=NOT _1X18;
PressInGvs_K5:=NOT _1X19;
PressOutWtr_K4:=NOT _1X20;
PressInWtr_K4:=NOT _1X21;
PresBefoWtrPrepar1:=NOT _1X22;
PresBefoWtrPrepar2:=NOT _1X23;
PressOutLoadGvs_K14:=NOT _1X24;
PressInLoadGvs_K14:=NOT _1X25;
//------Модуль А1.3----------------------------
PressPodachi:=REAL_TO_INT(AnalogSensers.LT_PT3.OUT);
PressObratki:=REAL_TO_INT(AnalogSensers.LT_PT4.OUT);
PressPodachiGvs:=REAL_TO_INT(AnalogSensers.LT_PT6.OUT);
PressObratkiGvs:=REAL_TO_INT(AnalogSensers.LT_PT5.OUT);
PressWtr:=REAL_TO_INT(AnalogSensers.LT_PT8.OUT);
PressGass:=REAL_TO_INT(AnalogSensers.LT_PT10.OUT);
//------Модуль А1.4----------------------------
TmpWtrInBoilerK8:=TE1;
TmpWtrIn1BoilerK2:=TE2;
TmpWtrIn2BoilerK2:=TE3;
TmpWtrPodachi:=TE4;
//------Модуль А1.5----------------------------
TmpWtrObratki:=TE5;
TmpWtrPodachiGvs:=TE6;
TmpWtrObratkiGvs:=TE7;
TmpAir:=TE8;
//------Модуль А1.6----------------------------
TmpWtrGvs:=TE9;

//--------Modbus ГВС чтение-------------------
CURRENT_GVS:=_CURRENT_GVS;
FREQUENSY_GVS:=_FREQUENSY_GVS/400;

//--------Modbus СЕТЕВОЙ 1чтение -------------------
CURRENT_NETWORK_1:=_CURRENT_NETWORK_1;
FREQUENSY_NETWORK_1:=_FREQUENSY_NETWORK_1/400;

//--------Modbus СЕТЕВОЙ 2 чтение-------------------
CURRENT_NETWORK_2:=_CURRENT_NETWORK_2;
FREQUENSY_NETWORK_2:=_FREQUENSY_NETWORK_2/400;

//--------Modbus ГВС запись-------------------
_KP_GVS:=KP_GVS;
_KI_GVS:=KI_GVS;
_KD_GVS:=KD_GVS;
_SET_POINT_GVS:=SET_POINT_GVS;

//--------Modbus СЕТЕВОЙ 1 запись -------------------	
_KP_NETWORK_1:=KP_NETWORK_1;
_KI_NETWORK_1:=KI_NETWORK_1;
_KD_NETWORK_1:=KD_NETWORK_1;
_SET_POINT_NETWORK_1:=SET_POINT_NETWORK_1;

//--------Modbus СЕТЕВОЙ 2 запись-------------------		
_KP_NETWORK_2:=KP_NETWORK_2;
_KI_NETWORK_2:=KI_NETWORK_2;
_KD_NETWORK_2:=KD_NETWORK_2;
_SET_POINT_NETWORK_2:=SET_POINT_NETWORK_2;

//--------Modbus BOILER 1 запись-------------------
IF HandModeBoiler1=TRUE THEN 
	_USTAVKA_TMP_CO_1:=USTAVKA_TMP_CO_1;
	ELSE
	_USTAVKA_TMP_CO_1:=PidMeteoVlv.GraficPodachi.OUT+10;
END_IF
CurrentUstavka1:=_USTAVKA_TMP_CO_1;
//--------Modbus BOILER 2 запись-------------------
IF HandModeBoiler2=TRUE THEN 
	_USTAVKA_TMP_CO_2:=USTAVKA_TMP_CO_2;
	ELSE
	_USTAVKA_TMP_CO_2:=PidMeteoVlv.GraficPodachi.OUT+10;
END_IF
CurrentUstavka2:=_USTAVKA_TMP_CO_2;
//StaitBoiler1:=Boiler1[0];
//TmpCoBoiler1:=Boiler1[1];
//TmpRecirculationBoiler1:=Boiler1[2];
//TmpFire1_Boiler1:=Boiler1[3];
//TmpFire2_Boiler1:=Boiler1[4];
//TmpShnek1_Boiler1:=Boiler1[5];
//TmpShnek2_Boiler1:=Boiler1[6];	
//ErrBoiler1:=Boiler1[7];

//StaitBoiler2:=Boiler2[0];
//TmpCoBoiler2:=Boiler2[1];
//TmpRecirculationBoiler2:=Boiler2[2];
//TmpFire1_Boiler2:=Boiler2[3];
//TmpFire2_Boiler2:=Boiler2[4];
//TmpShnek1_Boiler2:=Boiler2[5];
//TmpShnek2_Boiler2:=Boiler2[6];	
//ErrBoiler2:=Boiler2[7];

%MW66:=StaitBoiler1;
%MW67:=TmpCoBoiler1;
%MW68:=TmpRecirculationBoiler1;
%MW69:=TmpFire1_Boiler1;
%MW70:=TmpFire2_Boiler1;
%MW71:=TmpShnek1_Boiler1;
%MW72:=TmpShnek2_Boiler1;	
%MW73:=ErrBoiler1;
	
%MW74:=StaitBoiler2;
%MW75:=TmpCoBoiler2;
%MW76:=TmpRecirculationBoiler2;
%MW77:=TmpFire1_Boiler2;
%MW78:=TmpFire2_Boiler2;
%MW79:=TmpShnek1_Boiler2;
%MW80:=TmpShnek2_Boiler2;	
%mw81:=ErrBoiler2;

END_PROGRAM

// MyController/Application/AnalogSensers
PROGRAM AnalogSensers
VAR
	LT_PT3: LIN_TRAFO;
	LT_PT4: LIN_TRAFO;
	LT_PT5: LIN_TRAFO;
	LT_PT6: LIN_TRAFO;
	LT_PT8: LIN_TRAFO;
	LT_PT10: LIN_TRAFO;
END_VAR

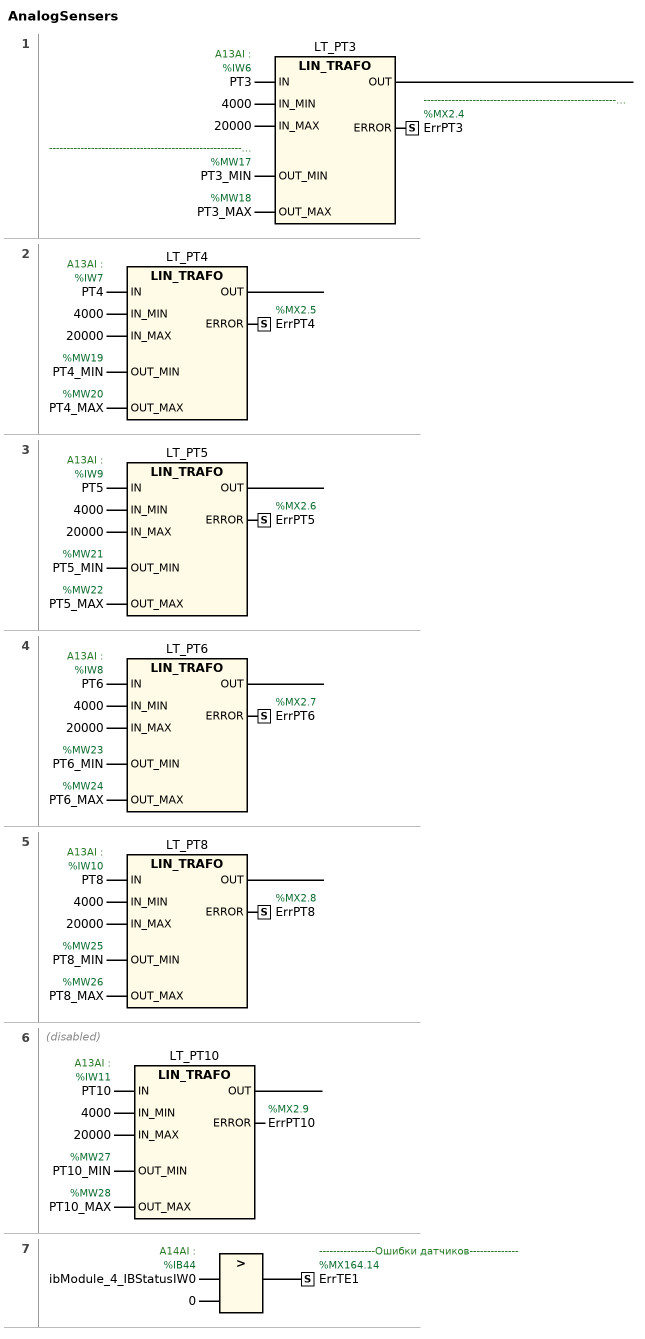
// NETWORK 1
//   PT3: A13AI : | AT %IW6
//   PT3_MIN: -------------------------------------------------------- -----AnalogSenser--------------------------------------- -------------------------------------------------------- | AT %MW17
//   PT3_MAX: AT %MW18
//   ErrPT3: -------------------------------------------------------- -----AnalogSensers----------------------------------------- -------------------------------------------------------- | AT %MX2.4
LT_PT3(IN := PT3, IN_MIN := 4000, IN_MAX := 20000, OUT_MIN := PT3_MIN, OUT_MAX := PT3_MAX); // LIN_TRAFO
ErrPT3 S= LT_PT3.ERROR;

// NETWORK 2
//   PT4: A13AI : | AT %IW7
//   PT4_MIN: AT %MW19
//   PT4_MAX: AT %MW20
//   ErrPT4: AT %MX2.5
LT_PT4(IN := PT4, IN_MIN := 4000, IN_MAX := 20000, OUT_MIN := PT4_MIN, OUT_MAX := PT4_MAX); // LIN_TRAFO
ErrPT4 S= LT_PT4.ERROR;

// NETWORK 3
//   PT5: A13AI : | AT %IW9
//   PT5_MIN: AT %MW21
//   PT5_MAX: AT %MW22
//   ErrPT5: AT %MX2.6
LT_PT5(IN := PT5, IN_MIN := 4000, IN_MAX := 20000, OUT_MIN := PT5_MIN, OUT_MAX := PT5_MAX); // LIN_TRAFO
ErrPT5 S= LT_PT5.ERROR;

// NETWORK 4
//   PT6: A13AI : | AT %IW8
//   PT6_MIN: AT %MW23
//   PT6_MAX: AT %MW24
//   ErrPT6: AT %MX2.7
LT_PT6(IN := PT6, IN_MIN := 4000, IN_MAX := 20000, OUT_MIN := PT6_MIN, OUT_MAX := PT6_MAX); // LIN_TRAFO
ErrPT6 S= LT_PT6.ERROR;

// NETWORK 5
//   PT8: A13AI : | AT %IW10
//   PT8_MIN: AT %MW25
//   PT8_MAX: AT %MW26
//   ErrPT8: AT %MX2.8
LT_PT8(IN := PT8, IN_MIN := 4000, IN_MAX := 20000, OUT_MIN := PT8_MIN, OUT_MAX := PT8_MAX); // LIN_TRAFO
ErrPT8 S= LT_PT8.ERROR;

// NETWORK 6 (disabled)
//   PT10: A13AI : | AT %IW11
//   PT10_MIN: AT %MW27
//   PT10_MAX: AT %MW28
//   ErrPT10: AT %MX2.9
// LT_PT10(
//     IN := PT10,
//     IN_MIN := 4000,
//     IN_MAX := 20000,
//     OUT_MIN := PT10_MIN,
//     OUT_MAX := PT10_MAX,
//     ERROR => ErrPT10); // LIN_TRAFO

// NETWORK 7
//   ibModule_4_IBStatusIW0: A14AI : | AT %IB44
//   ErrTE1: ----------------Ошибки датчиков-------------- | AT %MX164.14
ErrTE1 S= ibModule_4_IBStatusIW0 > 0;

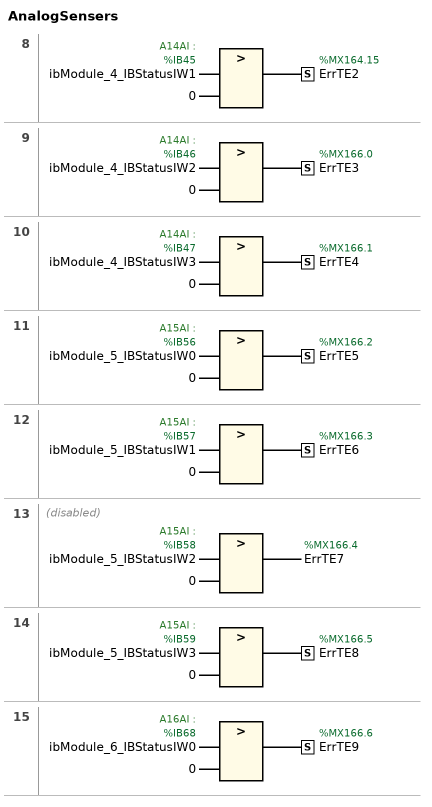
// NETWORK 8
//   ibModule_4_IBStatusIW1: A14AI : | AT %IB45
//   ErrTE2: AT %MX164.15
ErrTE2 S= ibModule_4_IBStatusIW1 > 0;

// NETWORK 9
//   ibModule_4_IBStatusIW2: A14AI : | AT %IB46
//   ErrTE3: AT %MX166.0
ErrTE3 S= ibModule_4_IBStatusIW2 > 0;

// NETWORK 10
//   ibModule_4_IBStatusIW3: A14AI : | AT %IB47
//   ErrTE4: AT %MX166.1
ErrTE4 S= ibModule_4_IBStatusIW3 > 0;

// NETWORK 11
//   ibModule_5_IBStatusIW0: A15AI : | AT %IB56
//   ErrTE5: AT %MX166.2
ErrTE5 S= ibModule_5_IBStatusIW0 > 0;

// NETWORK 12
//   ibModule_5_IBStatusIW1: A15AI : | AT %IB57
//   ErrTE6: AT %MX166.3
ErrTE6 S= ibModule_5_IBStatusIW1 > 0;

// NETWORK 13 (disabled)
//   ibModule_5_IBStatusIW2: A15AI : | AT %IB58
//   ErrTE7: AT %MX166.4
// ErrTE7 := ibModule_5_IBStatusIW2 > 0;

// NETWORK 14
//   ibModule_5_IBStatusIW3: A15AI : | AT %IB59
//   ErrTE8: AT %MX166.5
ErrTE8 S= ibModule_5_IBStatusIW3 > 0;

// NETWORK 15
//   ibModule_6_IBStatusIW0: A16AI : | AT %IB68
//   ErrTE9: AT %MX166.6
ErrTE9 S= ibModule_6_IBStatusIW0 > 0;

END_PROGRAM

// MyController/Application/PidMeteoVlv
PROGRAM PidMeteoVlv
VAR
	PID_Valve: PID;	
	DelayValveOpn: BLINK;
	DelayValveCls: BLINK;
	GraficPodachi: CHARCURVE;
	OutputLimit_TmpAir: OutputLimit;
	blink_1s: BLINK;
	BLINK2_1s: BLINK;
	InitializationTmpGrafik_Podachy: InitializationTmpGrafik;
END_VAR
VAR // added by the converter: edge detectors and wires of the graphical bodies
    _rt1, _rt2, _rt3, _rt4 : R_TRIG;
END_VAR

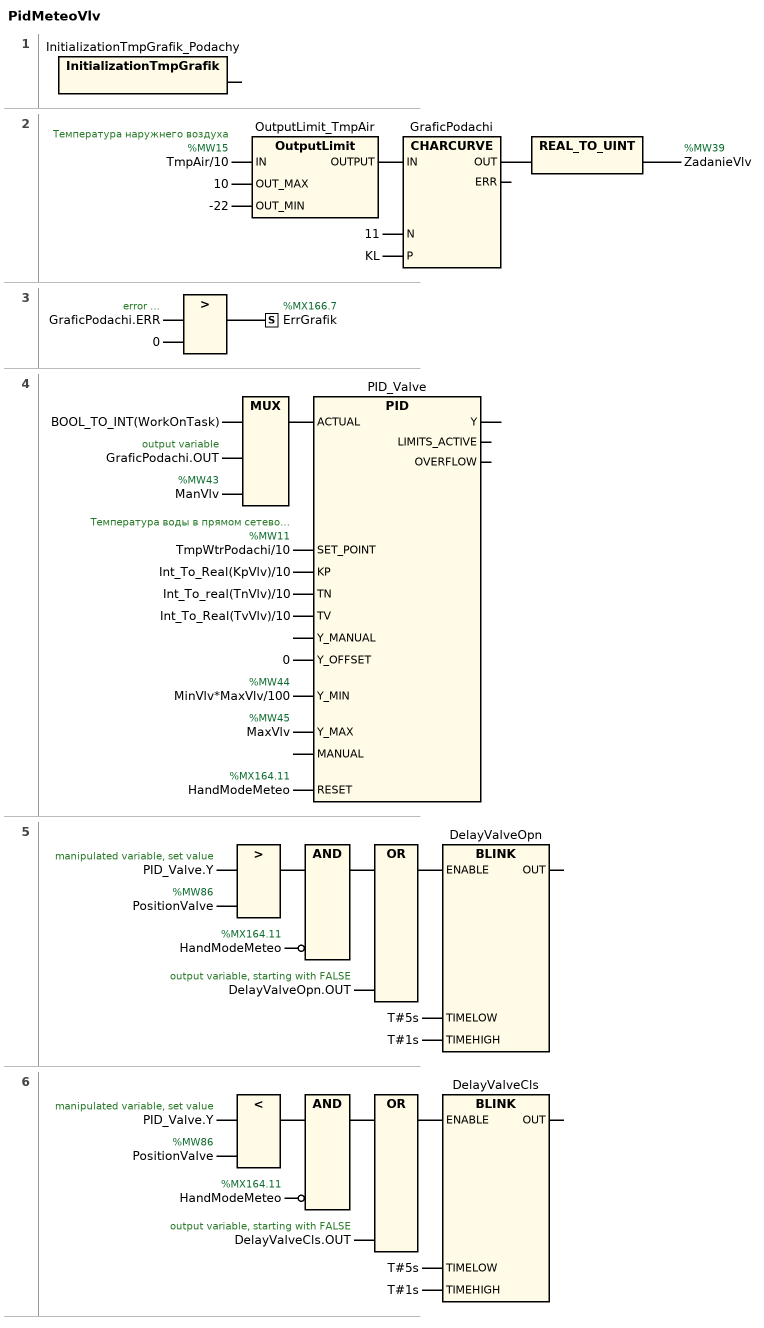
// NETWORK 1
InitializationTmpGrafik_Podachy(); // InitializationTmpGrafik

// NETWORK 2
//   TmpAir/10: Температура наружнего воздуха | AT %MW15
//   ZadanieVlv: AT %MW39
OutputLimit_TmpAir(IN := TmpAir/10, OUT_MAX := 10, OUT_MIN := -22); // OutputLimit
GraficPodachi(IN := OutputLimit_TmpAir.OUTPUT, N := 11, P := KL); // CHARCURVE
ZadanieVlv := REAL_TO_UINT(GraficPodachi.OUT);

// NETWORK 3
//   GraficPodachi.ERR: error : 0 : no error 1 : error in ARRAY: wrong sequence ( completely tested, only if IN is equal to largest X-value of P) 2 : IN outside of limits of P 4 : number of POINTS (N) invalid
//   ErrGrafik: AT %MX166.7
ErrGrafik S= GraficPodachi.ERR > 0;

// NETWORK 4
//   GraficPodachi.OUT: output variable
//   ManVlv: AT %MW43
//   TmpWtrPodachi/10: Температура воды в прямом сетевом трубопроводе на выходе из котельной (ТЕ4) | AT %MW11
//   MinVlv*MaxVlv/100: AT %MW44
//   MaxVlv: AT %MW45
//   HandModeMeteo: AT %MX164.11
PID_Valve(
    ACTUAL := MUX(BOOL_TO_INT(WorkOnTask), GraficPodachi.OUT, ManVlv),
    SET_POINT := TmpWtrPodachi/10,
    KP := Int_To_Real(KpVlv)/10,
    TN := Int_To_real(TnVlv)/10,
    TV := Int_To_Real(TvVlv)/10,
    Y_OFFSET := 0,
    Y_MIN := MinVlv*MaxVlv/100,
    Y_MAX := MaxVlv,
    RESET := HandModeMeteo); // PID

// NETWORK 5
//   PID_Valve.Y: manipulated variable, set value
//   PositionValve: AT %MW86
//   HandModeMeteo: AT %MX164.11
//   DelayValveOpn.OUT: output variable, starting with FALSE
DelayValveOpn(
    ENABLE := PID_Valve.Y > PositionValve AND NOT HandModeMeteo OR DelayValveOpn.OUT,
    TIMELOW := T#5s,
    TIMEHIGH := T#1s); // BLINK

// NETWORK 6
//   PID_Valve.Y: manipulated variable, set value
//   PositionValve: AT %MW86
//   HandModeMeteo: AT %MX164.11
//   DelayValveCls.OUT: output variable, starting with FALSE
DelayValveCls(
    ENABLE := PID_Valve.Y < PositionValve AND NOT HandModeMeteo OR DelayValveCls.OUT,
    TIMELOW := T#5s,
    TIMEHIGH := T#1s); // BLINK

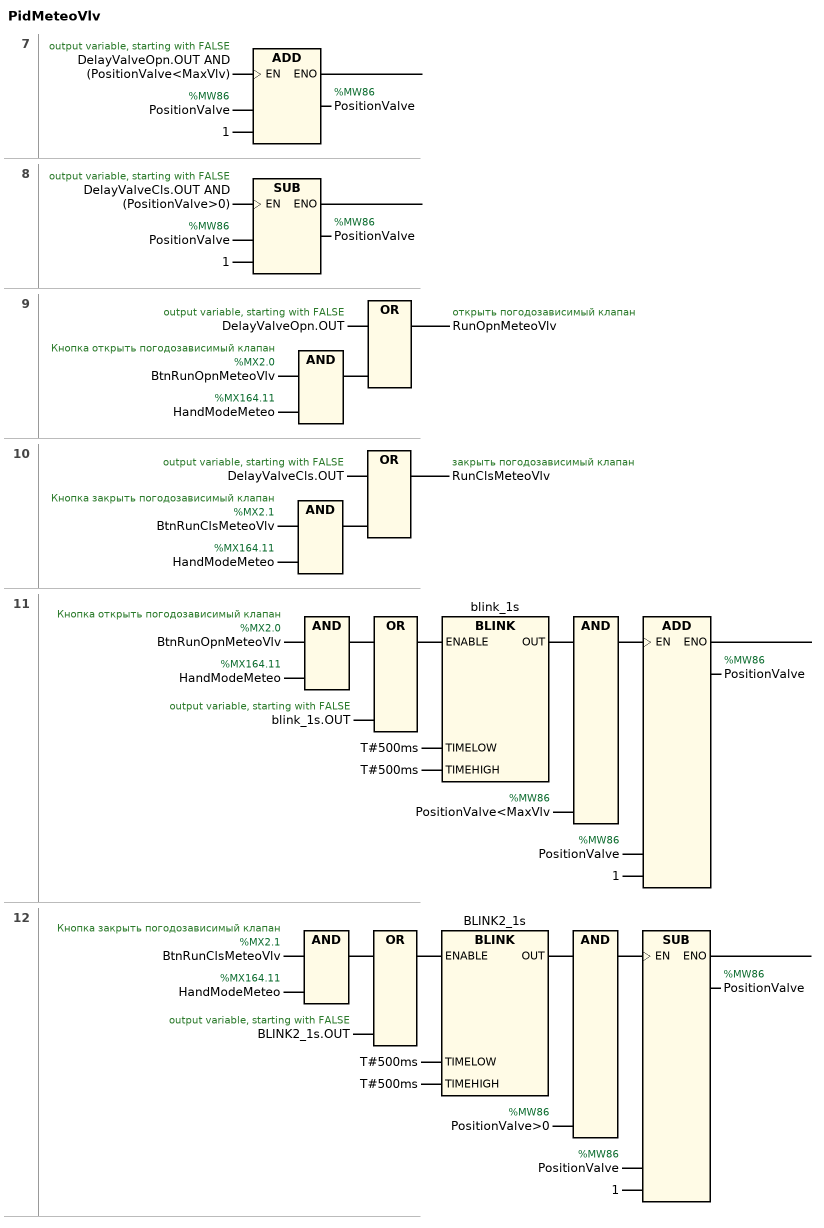
// NETWORK 7
//   DelayValveOpn.OUT AND (PositionValve<MaxVlv): output variable, starting with FALSE
//   PositionValve: AT %MW86
_rt1(CLK := DelayValveOpn.OUT AND (PositionValve<MaxVlv));
IF _rt1.Q THEN PositionValve := PositionValve + 1; END_IF

// NETWORK 8
//   DelayValveCls.OUT AND (PositionValve>0): output variable, starting with FALSE
//   PositionValve: AT %MW86
_rt2(CLK := DelayValveCls.OUT AND (PositionValve>0));
IF _rt2.Q THEN PositionValve := PositionValve - 1; END_IF

// NETWORK 9
//   DelayValveOpn.OUT: output variable, starting with FALSE
//   BtnRunOpnMeteoVlv: Кнопка открыть погодозависимый клапан | AT %MX2.0
//   HandModeMeteo: AT %MX164.11
//   RunOpnMeteoVlv: открыть погодозависимый клапан
RunOpnMeteoVlv := DelayValveOpn.OUT OR BtnRunOpnMeteoVlv AND HandModeMeteo;

// NETWORK 10
//   DelayValveCls.OUT: output variable, starting with FALSE
//   BtnRunClsMeteoVlv: Кнопка закрыть погодозависимый клапан | AT %MX2.1
//   HandModeMeteo: AT %MX164.11
//   RunClsMeteoVlv: закрыть погодозависимый клапан
RunClsMeteoVlv := DelayValveCls.OUT OR BtnRunClsMeteoVlv AND HandModeMeteo;

// NETWORK 11
//   BtnRunOpnMeteoVlv: Кнопка открыть погодозависимый клапан | AT %MX2.0
//   HandModeMeteo: AT %MX164.11
//   blink_1s.OUT: output variable, starting with FALSE
//   PositionValve<MaxVlv: AT %MW86
//   PositionValve: AT %MW86
blink_1s(
    ENABLE := BtnRunOpnMeteoVlv AND HandModeMeteo OR blink_1s.OUT,
    TIMELOW := T#500ms,
    TIMEHIGH := T#500ms); // BLINK
_rt3(CLK := blink_1s.OUT AND (PositionValve<MaxVlv));
IF _rt3.Q THEN PositionValve := PositionValve + 1; END_IF

// NETWORK 12
//   BtnRunClsMeteoVlv: Кнопка закрыть погодозависимый клапан | AT %MX2.1
//   HandModeMeteo: AT %MX164.11
//   BLINK2_1s.OUT: output variable, starting with FALSE
//   PositionValve>0: AT %MW86
//   PositionValve: AT %MW86
BLINK2_1s(
    ENABLE := BtnRunClsMeteoVlv AND HandModeMeteo OR BLINK2_1s.OUT,
    TIMELOW := T#500ms,
    TIMEHIGH := T#500ms); // BLINK
_rt4(CLK := BLINK2_1s.OUT AND (PositionValve>0));
IF _rt4.Q THEN PositionValve := PositionValve - 1; END_IF

END_PROGRAM

// MyController/Application/InitializationTmpGrafik
FUNCTION_BLOCK InitializationTmpGrafik
VAR_INPUT
END_VAR
VAR_OUTPUT
END_VAR
VAR
END_VAR

(*[(x:=-22,y:=84),
(x:=-19,y:=81),
(x:=-15,y:=76),
(x:=-13,y:=74),
(x:=-10,y:=71),
(x:=-7,y:=67),
(x:=-3,y:=63),
(x:=0,y:=60),
(x:=2,y:=58),
(x:=5,y:=55),
(x:=10,y:=55)];*)

KL[0].X:=-22;KL[0].Y:=TmpGrafN22;
KL[1].X:=-19;KL[1].Y:=TmpGrafN19;
KL[2].X:=-15;KL[2].Y:=TmpGrafN15;
KL[3].X:=-13;KL[3].Y:=TmpGrafN13;
KL[4].X:=-10;KL[4].Y:=TmpGrafN10;
KL[5].X:=-7;KL[5].Y:=TmpGrafN7;
KL[6].X:=-3;KL[6].Y:=TmpGrafN3;
KL[7].X:=0;KL[7].Y:=TmpGraf0;
KL[8].X:=2;KL[8].Y:=TmpGraf2;
KL[9].X:=5;KL[9].Y:=TmpGraf5;
KL[10].X:=10;KL[10].Y:=TmpGraf10;

END_FUNCTION_BLOCK

// MyController/Application/OutputLimit
FUNCTION_BLOCK OutputLimit
VAR_INPUT
	IN: INT;
	OUT_MAX: INT;
	OUT_MIN: INT;
END_VAR
VAR_OUTPUT
	OUTPUT: INT;
END_VAR
VAR
END_VAR

IF	IN>OUT_MAX THEN OUTPUT:=OUT_MAX;
ELSIF IN<OUT_MIN THEN OUTPUT:=OUT_MIN;
ELSE OUTPUT:=IN;
END_IF

END_FUNCTION_BLOCK

// MyController/Application/PidGvs
PROGRAM PidGvs
VAR
	PID_GvsValve: PID;
	DelayGvsValveOpn: BLINK;
	DelayGvsValveCls: BLINK;
	blink_gvs_1s: BLINK;
	BLINK2_GVS_1s: BLINK;
END_VAR
VAR // added by the converter: edge detectors and wires of the graphical bodies
    _rt1, _rt2, _rt3, _rt4 : R_TRIG;
END_VAR

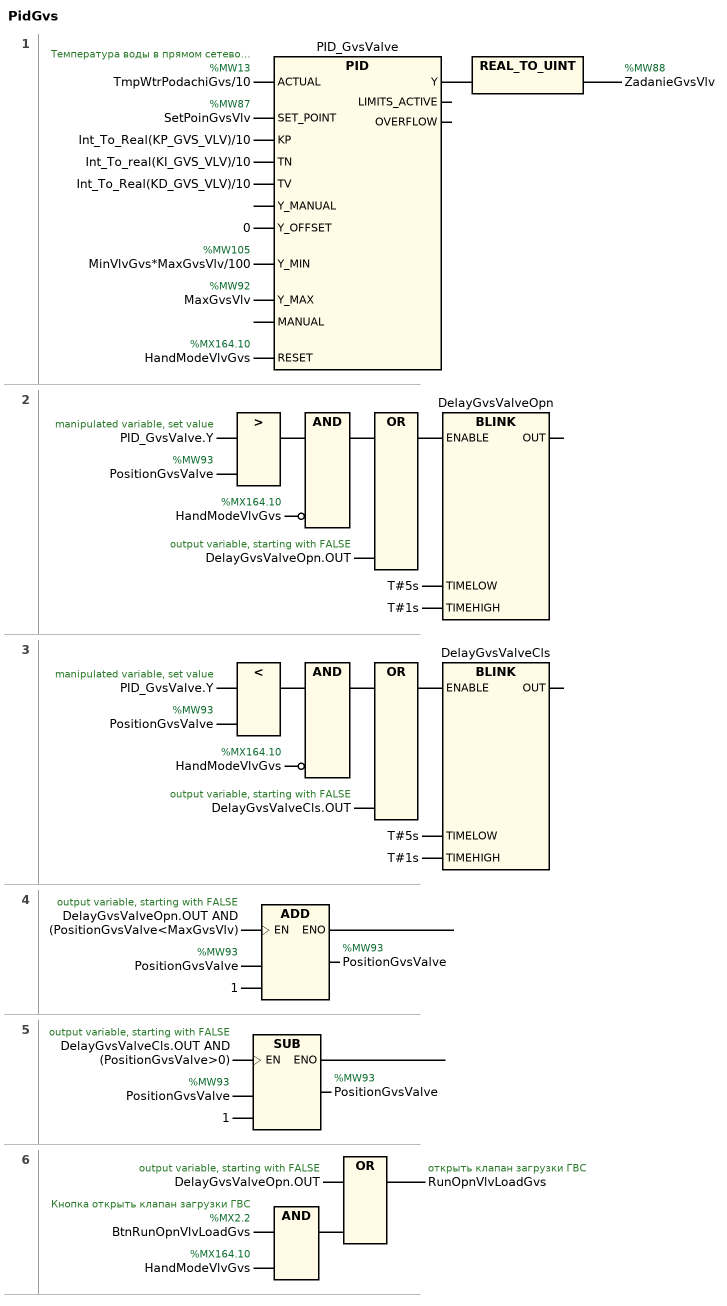
// NETWORK 1
//   TmpWtrPodachiGvs/10: Температура воды в прямом сетевом трубопроводе ГВС на выходе из котельной (ТЕ6) | AT %MW13
//   SetPoinGvsVlv: AT %MW87
//   MinVlvGvs*MaxGvsVlv/100: AT %MW105
//   MaxGvsVlv: AT %MW92
//   HandModeVlvGvs: AT %MX164.10
//   ZadanieGvsVlv: AT %MW88
PID_GvsValve(
    ACTUAL := TmpWtrPodachiGvs/10,
    SET_POINT := SetPoinGvsVlv,
    KP := Int_To_Real(KP_GVS_VLV)/10,
    TN := Int_To_real(KI_GVS_VLV)/10,
    TV := Int_To_Real(KD_GVS_VLV)/10,
    Y_OFFSET := 0,
    Y_MIN := MinVlvGvs*MaxGvsVlv/100,
    Y_MAX := MaxGvsVlv,
    RESET := HandModeVlvGvs); // PID
ZadanieGvsVlv := REAL_TO_UINT(PID_GvsValve.Y);

// NETWORK 2
//   PID_GvsValve.Y: manipulated variable, set value
//   PositionGvsValve: AT %MW93
//   HandModeVlvGvs: AT %MX164.10
//   DelayGvsValveOpn.OUT: output variable, starting with FALSE
DelayGvsValveOpn(
    ENABLE := PID_GvsValve.Y > PositionGvsValve AND NOT HandModeVlvGvs OR DelayGvsValveOpn.OUT,
    TIMELOW := T#5s,
    TIMEHIGH := T#1s); // BLINK

// NETWORK 3
//   PID_GvsValve.Y: manipulated variable, set value
//   PositionGvsValve: AT %MW93
//   HandModeVlvGvs: AT %MX164.10
//   DelayGvsValveCls.OUT: output variable, starting with FALSE
DelayGvsValveCls(
    ENABLE := PID_GvsValve.Y < PositionGvsValve AND NOT HandModeVlvGvs OR DelayGvsValveCls.OUT,
    TIMELOW := T#5s,
    TIMEHIGH := T#1s); // BLINK

// NETWORK 4
//   DelayGvsValveOpn.OUT AND (PositionGvsValve<MaxGvsVlv): output variable, starting with FALSE
//   PositionGvsValve: AT %MW93
_rt1(CLK := DelayGvsValveOpn.OUT AND (PositionGvsValve<MaxGvsVlv));
IF _rt1.Q THEN PositionGvsValve := PositionGvsValve + 1; END_IF

// NETWORK 5
//   DelayGvsValveCls.OUT AND (PositionGvsValve>0): output variable, starting with FALSE
//   PositionGvsValve: AT %MW93
_rt2(CLK := DelayGvsValveCls.OUT AND (PositionGvsValve>0));
IF _rt2.Q THEN PositionGvsValve := PositionGvsValve - 1; END_IF

// NETWORK 6
//   DelayGvsValveOpn.OUT: output variable, starting with FALSE
//   BtnRunOpnVlvLoadGvs: Кнопка открыть клапан загрузки ГВС | AT %MX2.2
//   HandModeVlvGvs: AT %MX164.10
//   RunOpnVlvLoadGvs: открыть клапан загрузки ГВС
RunOpnVlvLoadGvs := DelayGvsValveOpn.OUT OR BtnRunOpnVlvLoadGvs AND HandModeVlvGvs;

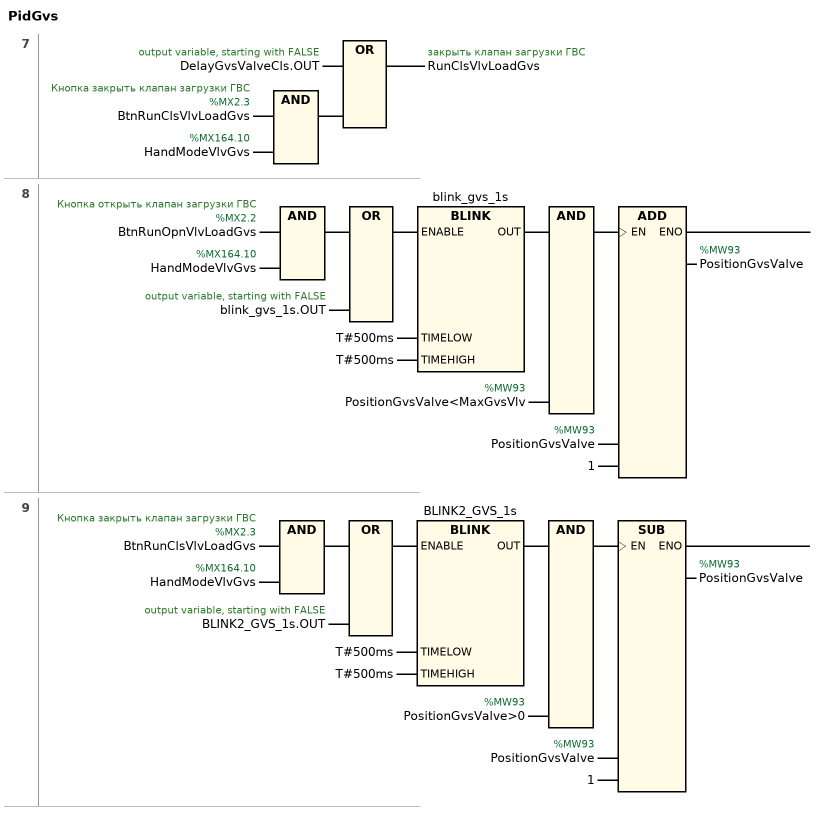
// NETWORK 7
//   DelayGvsValveCls.OUT: output variable, starting with FALSE
//   BtnRunClsVlvLoadGvs: Кнопка закрыть клапан загрузки ГВС | AT %MX2.3
//   HandModeVlvGvs: AT %MX164.10
//   RunClsVlvLoadGvs: закрыть клапан загрузки ГВС
RunClsVlvLoadGvs := DelayGvsValveCls.OUT OR BtnRunClsVlvLoadGvs AND HandModeVlvGvs;

// NETWORK 8
//   BtnRunOpnVlvLoadGvs: Кнопка открыть клапан загрузки ГВС | AT %MX2.2
//   HandModeVlvGvs: AT %MX164.10
//   blink_gvs_1s.OUT: output variable, starting with FALSE
//   PositionGvsValve<MaxGvsVlv: AT %MW93
//   PositionGvsValve: AT %MW93
blink_gvs_1s(
    ENABLE := BtnRunOpnVlvLoadGvs AND HandModeVlvGvs OR blink_gvs_1s.OUT,
    TIMELOW := T#500ms,
    TIMEHIGH := T#500ms); // BLINK
_rt3(CLK := blink_gvs_1s.OUT AND (PositionGvsValve<MaxGvsVlv));
IF _rt3.Q THEN PositionGvsValve := PositionGvsValve + 1; END_IF

// NETWORK 9
//   BtnRunClsVlvLoadGvs: Кнопка закрыть клапан загрузки ГВС | AT %MX2.3
//   HandModeVlvGvs: AT %MX164.10
//   BLINK2_GVS_1s.OUT: output variable, starting with FALSE
//   PositionGvsValve>0: AT %MW93
//   PositionGvsValve: AT %MW93
BLINK2_GVS_1s(
    ENABLE := BtnRunClsVlvLoadGvs AND HandModeVlvGvs OR BLINK2_GVS_1s.OUT,
    TIMELOW := T#500ms,
    TIMEHIGH := T#500ms); // BLINK
_rt4(CLK := BLINK2_GVS_1s.OUT AND (PositionGvsValve>0));
IF _rt4.Q THEN PositionGvsValve := PositionGvsValve - 1; END_IF

END_PROGRAM

// MyController/Application/ManualMode
PROGRAM ManualMode
VAR
	BLINK_Siren: BLINK;
	TM1: TOF;
	TM2: TOF;
	tm_reset_btn: TON;
	tm_reset_err: TON;
	tm_run_rec3: TON;
	tm_reset_btn_rcr3: TON;
	ReadDataFromGrands: SendData;
	var1: word_real;
END_VAR
VAR // added by the converter: edge detectors and wires of the graphical bodies
    _rt1, _rt2 : R_TRIG;
    _w1, _w2, _w3, _w4, _w5, _w6, _w7 : BOOL;
    _ft1, _ft2 : F_TRIG;
END_VAR

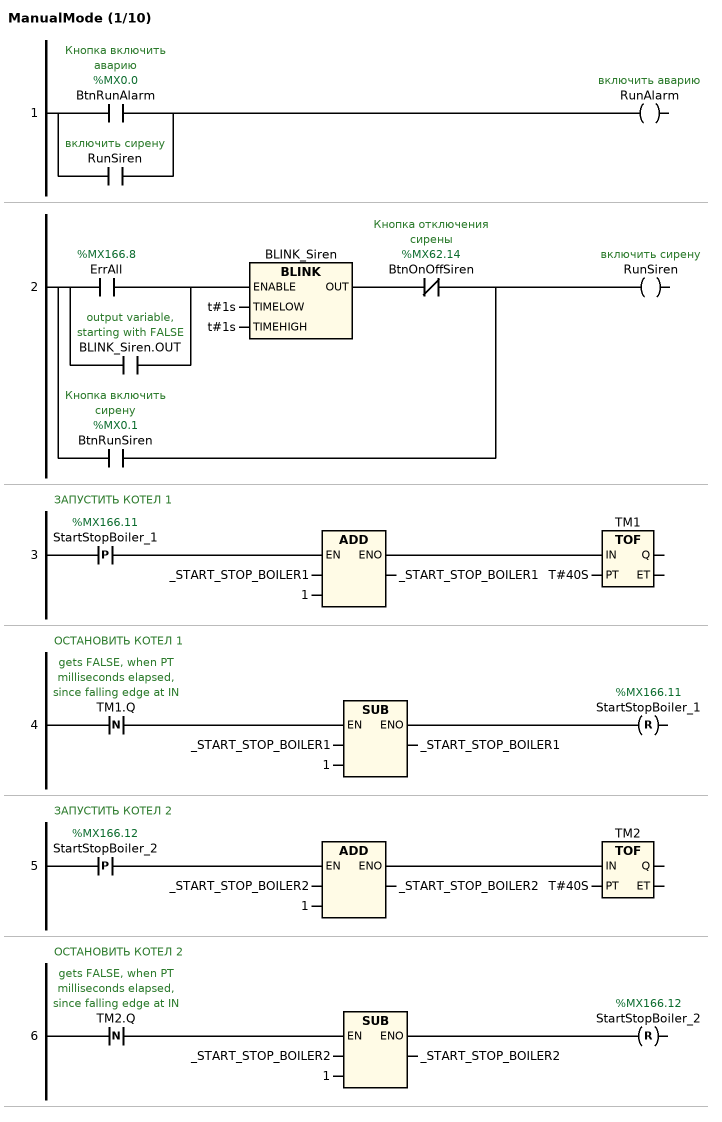
// NETWORK 1
//   BtnRunAlarm: Кнопка включить аварию | AT %MX0.0
//   RunSiren: включить сирену
//   RunAlarm: включить аварию
RunAlarm := BtnRunAlarm OR RunSiren;

// NETWORK 2
//   ErrAll: AT %MX166.8
//   BLINK_Siren.OUT: output variable, starting with FALSE
//   BtnOnOffSiren: Кнопка отключения сирены | AT %MX62.14
//   BtnRunSiren: Кнопка включить сирену | AT %MX0.1
//   RunSiren: включить сирену
BLINK_Siren(ENABLE := ErrAll OR BLINK_Siren.OUT, TIMELOW := t#1s, TIMEHIGH := t#1s); // BLINK
RunSiren := BLINK_Siren.OUT AND NOT BtnOnOffSiren OR BtnRunSiren;

// NETWORK 3
// ЗАПУСТИТЬ КОТЕЛ 1
//   StartStopBoiler_1: AT %MX166.11
_rt1(CLK := StartStopBoiler_1);
_w1 := _rt1.Q;
IF _w1 THEN _START_STOP_BOILER1 := _START_STOP_BOILER1 + 1; END_IF
TM1(IN := _w1, PT := T#40S); // TOF

// NETWORK 4
// ОСТАНОВИТЬ КОТЕЛ 1
//   TM1.Q: gets FALSE, when PT milliseconds elapsed, since falling edge at IN
//   StartStopBoiler_1: AT %MX166.11
_ft1(CLK := TM1.Q);
_w2 := _ft1.Q;
IF _w2 THEN _START_STOP_BOILER1 := _START_STOP_BOILER1 - 1; END_IF
StartStopBoiler_1 R= _w2;

// NETWORK 5
// ЗАПУСТИТЬ КОТЕЛ 2
//   StartStopBoiler_2: AT %MX166.12
_rt2(CLK := StartStopBoiler_2);
_w3 := _rt2.Q;
IF _w3 THEN _START_STOP_BOILER2 := _START_STOP_BOILER2 + 1; END_IF
TM2(IN := _w3, PT := T#40S); // TOF

// NETWORK 6
// ОСТАНОВИТЬ КОТЕЛ 2
//   TM2.Q: gets FALSE, when PT milliseconds elapsed, since falling edge at IN
//   StartStopBoiler_2: AT %MX166.12
_ft2(CLK := TM2.Q);
_w4 := _ft2.Q;
IF _w4 THEN _START_STOP_BOILER2 := _START_STOP_BOILER2 - 1; END_IF
StartStopBoiler_2 R= _w4;

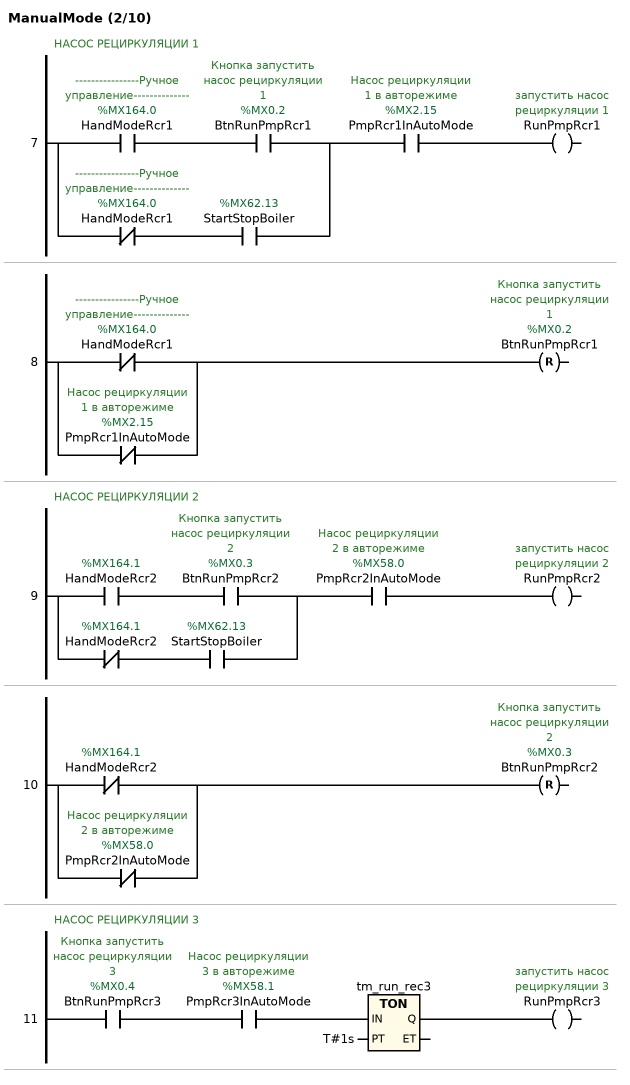
// NETWORK 7
// НАСОС РЕЦИРКУЛЯЦИИ 1
//   HandModeRcr1: ----------------Ручное управление-------------- | AT %MX164.0
//   BtnRunPmpRcr1: Кнопка запустить насос рециркуляции 1 | AT %MX0.2
//   StartStopBoiler: AT %MX62.13
//   PmpRcr1InAutoMode: Насос рециркуляции 1 в авторежиме | AT %MX2.15
//   RunPmpRcr1: запустить насос рециркуляции 1
RunPmpRcr1 := (HandModeRcr1 AND BtnRunPmpRcr1 OR NOT HandModeRcr1 AND StartStopBoiler) AND PmpRcr1InAutoMode;

// NETWORK 8
//   HandModeRcr1: ----------------Ручное управление-------------- | AT %MX164.0
//   PmpRcr1InAutoMode: Насос рециркуляции 1 в авторежиме | AT %MX2.15
//   BtnRunPmpRcr1: Кнопка запустить насос рециркуляции 1 | AT %MX0.2
BtnRunPmpRcr1 R= NOT HandModeRcr1 OR NOT PmpRcr1InAutoMode;

// NETWORK 9
// НАСОС РЕЦИРКУЛЯЦИИ 2
//   HandModeRcr2: AT %MX164.1
//   BtnRunPmpRcr2: Кнопка запустить насос рециркуляции 2 | AT %MX0.3
//   StartStopBoiler: AT %MX62.13
//   PmpRcr2InAutoMode: Насос рециркуляции 2 в авторежиме | AT %MX58.0
//   RunPmpRcr2: запустить насос рециркуляции 2
RunPmpRcr2 := (HandModeRcr2 AND BtnRunPmpRcr2 OR NOT HandModeRcr2 AND StartStopBoiler) AND PmpRcr2InAutoMode;

// NETWORK 10
//   HandModeRcr2: AT %MX164.1
//   PmpRcr2InAutoMode: Насос рециркуляции 2 в авторежиме | AT %MX58.0
//   BtnRunPmpRcr2: Кнопка запустить насос рециркуляции 2 | AT %MX0.3
BtnRunPmpRcr2 R= NOT HandModeRcr2 OR NOT PmpRcr2InAutoMode;

// NETWORK 11
// НАСОС РЕЦИРКУЛЯЦИИ 3
//   BtnRunPmpRcr3: Кнопка запустить насос рециркуляции 3 | AT %MX0.4
//   PmpRcr3InAutoMode: Насос рециркуляции 3 в авторежиме | AT %MX58.1
//   RunPmpRcr3: запустить насос рециркуляции 3
tm_run_rec3(IN := BtnRunPmpRcr3 AND PmpRcr3InAutoMode, PT := T#1s); // TON
RunPmpRcr3 := tm_run_rec3.Q;

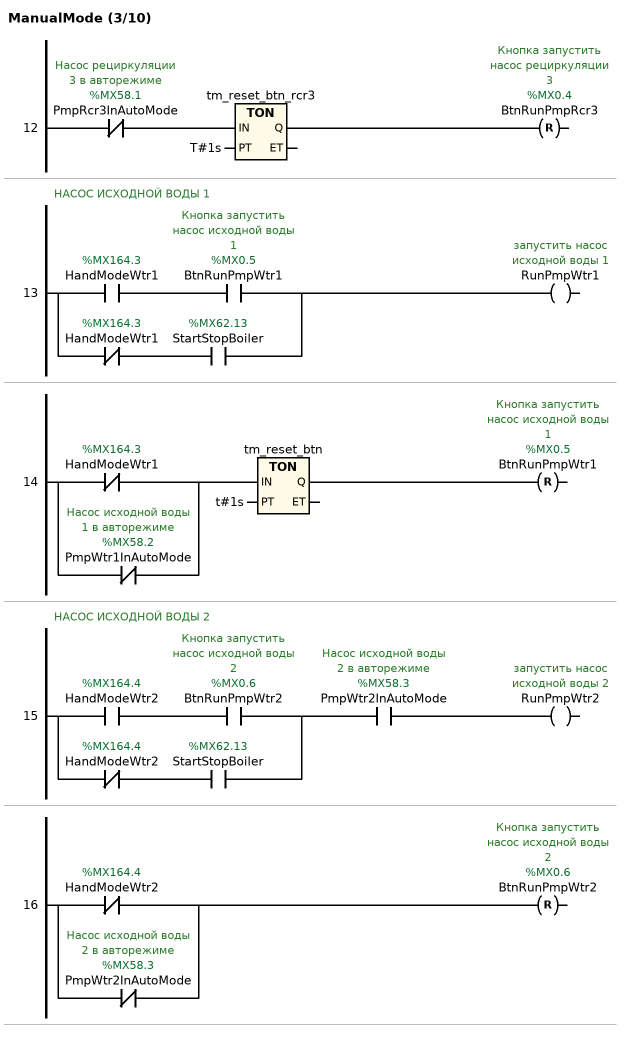
// NETWORK 12
//   PmpRcr3InAutoMode: Насос рециркуляции 3 в авторежиме | AT %MX58.1
//   BtnRunPmpRcr3: Кнопка запустить насос рециркуляции 3 | AT %MX0.4
tm_reset_btn_rcr3(IN := NOT PmpRcr3InAutoMode, PT := T#1s); // TON
BtnRunPmpRcr3 R= tm_reset_btn_rcr3.Q;

// NETWORK 13
// НАСОС ИСХОДНОЙ ВОДЫ 1
//   HandModeWtr1: AT %MX164.3
//   BtnRunPmpWtr1: Кнопка запустить насос исходной воды 1 | AT %MX0.5
//   StartStopBoiler: AT %MX62.13
//   RunPmpWtr1: запустить насос исходной воды 1
RunPmpWtr1 := HandModeWtr1 AND BtnRunPmpWtr1 OR NOT HandModeWtr1 AND StartStopBoiler;

// NETWORK 14
//   HandModeWtr1: AT %MX164.3
//   PmpWtr1InAutoMode: Насос исходной воды 1 в авторежиме | AT %MX58.2
//   BtnRunPmpWtr1: Кнопка запустить насос исходной воды 1 | AT %MX0.5
tm_reset_btn(IN := NOT HandModeWtr1 OR NOT PmpWtr1InAutoMode, PT := t#1s); // TON
BtnRunPmpWtr1 R= tm_reset_btn.Q;

// NETWORK 15
// НАСОС ИСХОДНОЙ ВОДЫ 2
//   HandModeWtr2: AT %MX164.4
//   BtnRunPmpWtr2: Кнопка запустить насос исходной воды 2 | AT %MX0.6
//   StartStopBoiler: AT %MX62.13
//   PmpWtr2InAutoMode: Насос исходной воды 2 в авторежиме | AT %MX58.3
//   RunPmpWtr2: запустить насос исходной воды 2
RunPmpWtr2 := (HandModeWtr2 AND BtnRunPmpWtr2 OR NOT HandModeWtr2 AND StartStopBoiler) AND PmpWtr2InAutoMode;

// NETWORK 16
//   HandModeWtr2: AT %MX164.4
//   PmpWtr2InAutoMode: Насос исходной воды 2 в авторежиме | AT %MX58.3
//   BtnRunPmpWtr2: Кнопка запустить насос исходной воды 2 | AT %MX0.6
BtnRunPmpWtr2 R= NOT HandModeWtr2 OR NOT PmpWtr2InAutoMode;

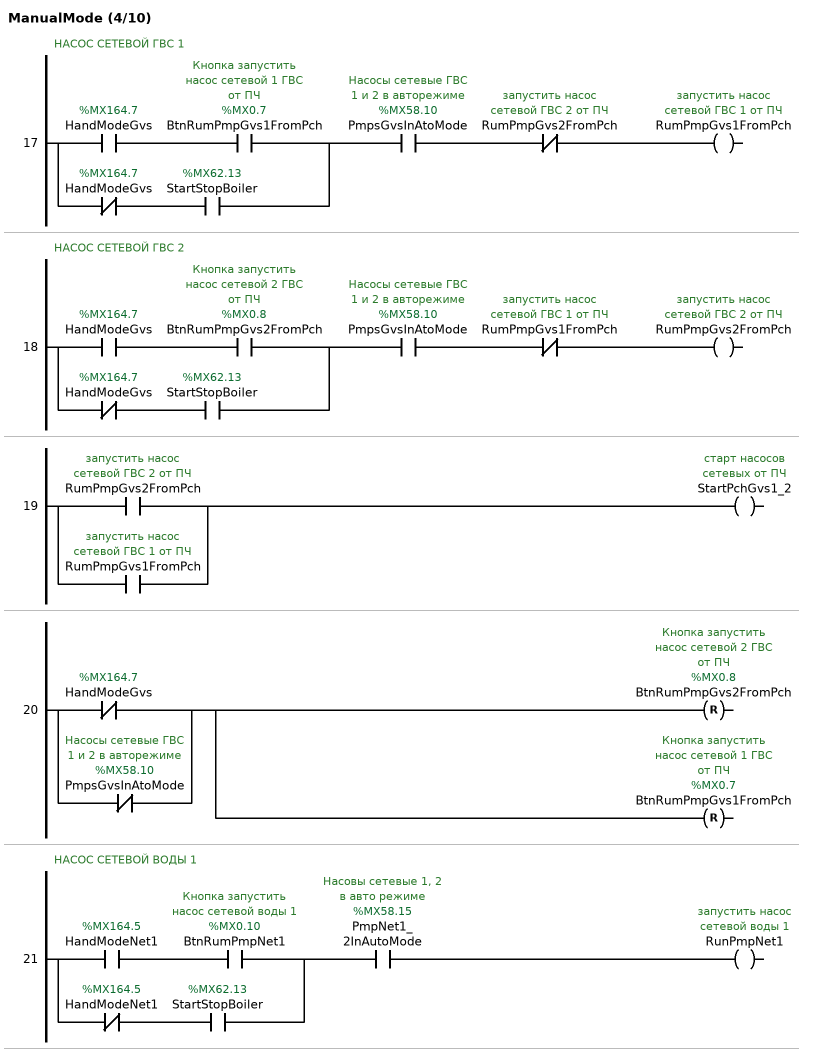
// NETWORK 17
// НАСОС СЕТЕВОЙ ГВС 1
//   HandModeGvs: AT %MX164.7
//   BtnRumPmpGvs1FromPch: Кнопка запустить насос сетевой 1 ГВС от ПЧ | AT %MX0.7
//   StartStopBoiler: AT %MX62.13
//   PmpsGvsInAtoMode: Насосы сетевые ГВС 1 и 2 в авторежиме | AT %MX58.10
//   RumPmpGvs2FromPch: запустить насос сетевой ГВС 2 от ПЧ
//   RumPmpGvs1FromPch: запустить насос сетевой ГВС 1 от ПЧ
RumPmpGvs1FromPch := (HandModeGvs AND BtnRumPmpGvs1FromPch OR NOT HandModeGvs AND StartStopBoiler) AND PmpsGvsInAtoMode AND NOT RumPmpGvs2FromPch;

// NETWORK 18
// НАСОС СЕТЕВОЙ ГВС 2
//   HandModeGvs: AT %MX164.7
//   BtnRumPmpGvs2FromPch: Кнопка запустить насос сетевой 2 ГВС от ПЧ | AT %MX0.8
//   StartStopBoiler: AT %MX62.13
//   PmpsGvsInAtoMode: Насосы сетевые ГВС 1 и 2 в авторежиме | AT %MX58.10
//   RumPmpGvs1FromPch: запустить насос сетевой ГВС 1 от ПЧ
//   RumPmpGvs2FromPch: запустить насос сетевой ГВС 2 от ПЧ
RumPmpGvs2FromPch := (HandModeGvs AND BtnRumPmpGvs2FromPch OR NOT HandModeGvs AND StartStopBoiler) AND PmpsGvsInAtoMode AND NOT RumPmpGvs1FromPch;

// NETWORK 19
//   RumPmpGvs2FromPch: запустить насос сетевой ГВС 2 от ПЧ
//   RumPmpGvs1FromPch: запустить насос сетевой ГВС 1 от ПЧ
//   StartPchGvs1_2: старт насосов сетевых от ПЧ
StartPchGvs1_2 := RumPmpGvs2FromPch OR RumPmpGvs1FromPch;

// NETWORK 20
//   HandModeGvs: AT %MX164.7
//   PmpsGvsInAtoMode: Насосы сетевые ГВС 1 и 2 в авторежиме | AT %MX58.10
//   BtnRumPmpGvs2FromPch: Кнопка запустить насос сетевой 2 ГВС от ПЧ | AT %MX0.8
//   BtnRumPmpGvs1FromPch: Кнопка запустить насос сетевой 1 ГВС от ПЧ | AT %MX0.7
_w5 := NOT HandModeGvs OR NOT PmpsGvsInAtoMode;
BtnRumPmpGvs2FromPch R= _w5;
BtnRumPmpGvs1FromPch R= _w5;

// NETWORK 21
// НАСОС СЕТЕВОЙ ВОДЫ 1
//   HandModeNet1: AT %MX164.5
//   BtnRumPmpNet1: Кнопка запустить насос сетевой воды 1 | AT %MX0.10
//   StartStopBoiler: AT %MX62.13
//   PmpNet1_2InAutoMode: Насовы сетевые 1, 2 в авто режиме | AT %MX58.15
//   RunPmpNet1: запустить насос сетевой воды 1
RunPmpNet1 := (HandModeNet1 AND BtnRumPmpNet1 OR NOT HandModeNet1 AND StartStopBoiler) AND PmpNet1_2InAutoMode;

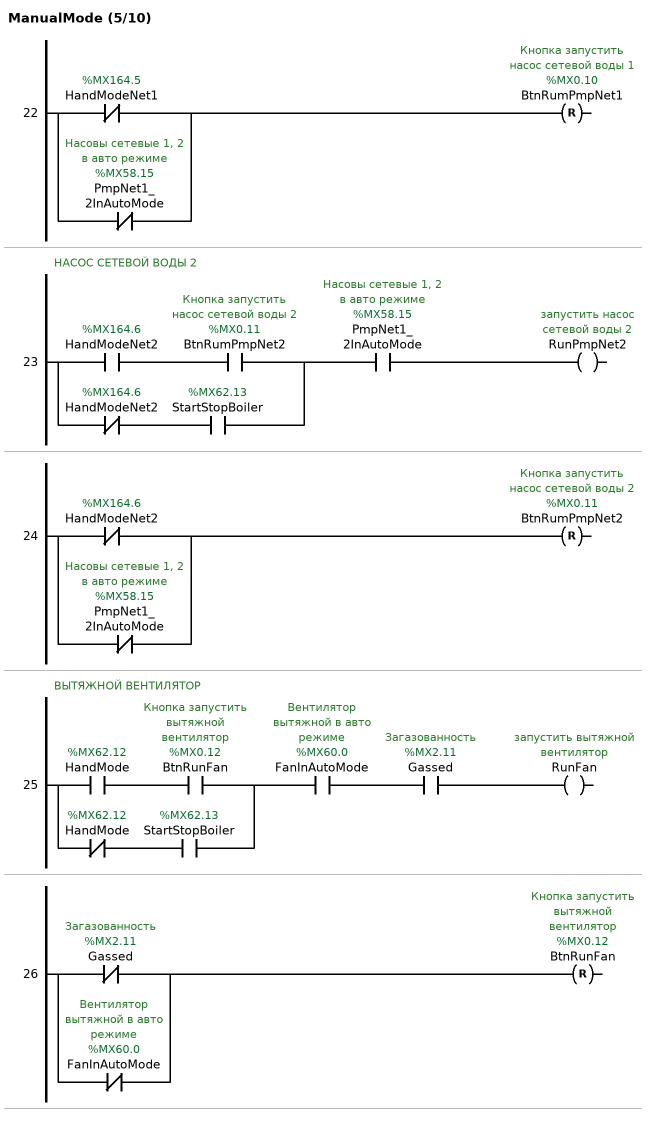
// NETWORK 22
//   HandModeNet1: AT %MX164.5
//   PmpNet1_2InAutoMode: Насовы сетевые 1, 2 в авто режиме | AT %MX58.15
//   BtnRumPmpNet1: Кнопка запустить насос сетевой воды 1 | AT %MX0.10
BtnRumPmpNet1 R= NOT HandModeNet1 OR NOT PmpNet1_2InAutoMode;

// NETWORK 23
// НАСОС СЕТЕВОЙ ВОДЫ 2
//   HandModeNet2: AT %MX164.6
//   BtnRumPmpNet2: Кнопка запустить насос сетевой воды 2 | AT %MX0.11
//   StartStopBoiler: AT %MX62.13
//   PmpNet1_2InAutoMode: Насовы сетевые 1, 2 в авто режиме | AT %MX58.15
//   RunPmpNet2: запустить насос сетевой воды 2
RunPmpNet2 := (HandModeNet2 AND BtnRumPmpNet2 OR NOT HandModeNet2 AND StartStopBoiler) AND PmpNet1_2InAutoMode;

// NETWORK 24
//   HandModeNet2: AT %MX164.6
//   PmpNet1_2InAutoMode: Насовы сетевые 1, 2 в авто режиме | AT %MX58.15
//   BtnRumPmpNet2: Кнопка запустить насос сетевой воды 2 | AT %MX0.11
BtnRumPmpNet2 R= NOT HandModeNet2 OR NOT PmpNet1_2InAutoMode;

// NETWORK 25
// ВЫТЯЖНОЙ ВЕНТИЛЯТОР
//   HandMode: AT %MX62.12
//   BtnRunFan: Кнопка запустить вытяжной вентилятор | AT %MX0.12
//   StartStopBoiler: AT %MX62.13
//   FanInAutoMode: Вентилятор вытяжной в авто режиме | AT %MX60.0
//   Gassed: Загазованность | AT %MX2.11
//   RunFan: запустить вытяжной вентилятор
RunFan := (HandMode AND BtnRunFan OR NOT HandMode AND StartStopBoiler) AND FanInAutoMode AND Gassed;

// NETWORK 26
//   Gassed: Загазованность | AT %MX2.11
//   FanInAutoMode: Вентилятор вытяжной в авто режиме | AT %MX60.0
//   BtnRunFan: Кнопка запустить вытяжной вентилятор | AT %MX0.12
BtnRunFan R= NOT Gassed OR NOT FanInAutoMode;

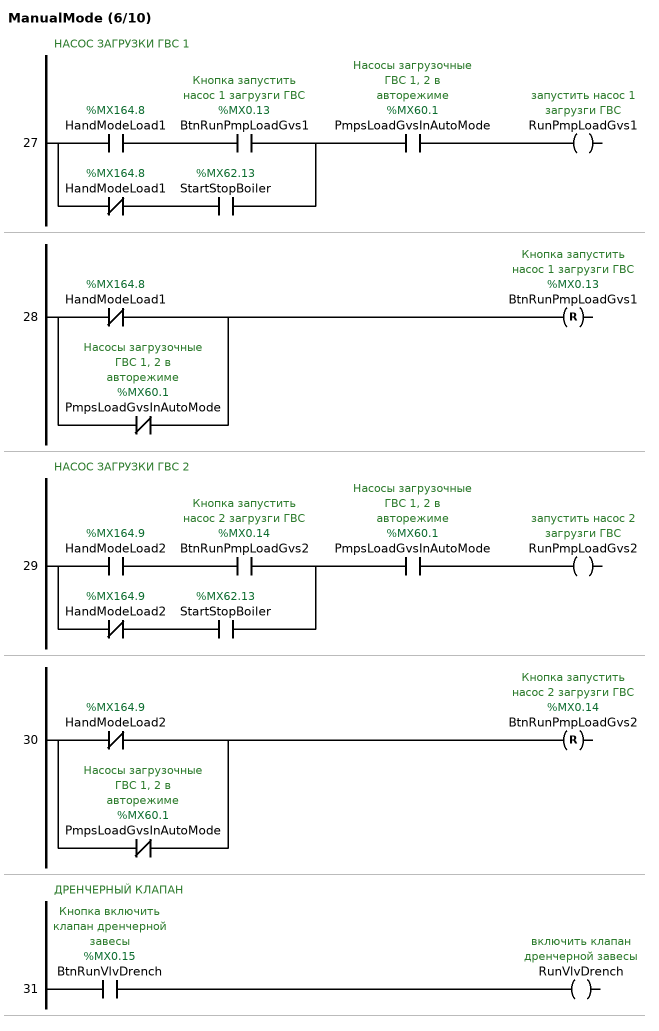
// NETWORK 27
// НАСОС ЗАГРУЗКИ ГВС 1
//   HandModeLoad1: AT %MX164.8
//   BtnRunPmpLoadGvs1: Кнопка запустить насос 1 загрузги ГВС | AT %MX0.13
//   StartStopBoiler: AT %MX62.13
//   PmpsLoadGvsInAutoMode: Насосы загрузочные ГВС 1, 2 в авторежиме | AT %MX60.1
//   RunPmpLoadGvs1: запустить насос 1 загрузги ГВС
RunPmpLoadGvs1 := (HandModeLoad1 AND BtnRunPmpLoadGvs1 OR NOT HandModeLoad1 AND StartStopBoiler) AND PmpsLoadGvsInAutoMode;

// NETWORK 28
//   HandModeLoad1: AT %MX164.8
//   PmpsLoadGvsInAutoMode: Насосы загрузочные ГВС 1, 2 в авторежиме | AT %MX60.1
//   BtnRunPmpLoadGvs1: Кнопка запустить насос 1 загрузги ГВС | AT %MX0.13
BtnRunPmpLoadGvs1 R= NOT HandModeLoad1 OR NOT PmpsLoadGvsInAutoMode;

// NETWORK 29
// НАСОС ЗАГРУЗКИ ГВС 2
//   HandModeLoad2: AT %MX164.9
//   BtnRunPmpLoadGvs2: Кнопка запустить насос 2 загрузги ГВС | AT %MX0.14
//   StartStopBoiler: AT %MX62.13
//   PmpsLoadGvsInAutoMode: Насосы загрузочные ГВС 1, 2 в авторежиме | AT %MX60.1
//   RunPmpLoadGvs2: запустить насос 2 загрузги ГВС
RunPmpLoadGvs2 := (HandModeLoad2 AND BtnRunPmpLoadGvs2 OR NOT HandModeLoad2 AND StartStopBoiler) AND PmpsLoadGvsInAutoMode;

// NETWORK 30
//   HandModeLoad2: AT %MX164.9
//   PmpsLoadGvsInAutoMode: Насосы загрузочные ГВС 1, 2 в авторежиме | AT %MX60.1
//   BtnRunPmpLoadGvs2: Кнопка запустить насос 2 загрузги ГВС | AT %MX0.14
BtnRunPmpLoadGvs2 R= NOT HandModeLoad2 OR NOT PmpsLoadGvsInAutoMode;

// NETWORK 31
// ДРЕНЧЕРНЫЙ КЛАПАН
//   BtnRunVlvDrench: Кнопка включить клапан дренчерной завесы | AT %MX0.15
//   RunVlvDrench: включить клапан дренчерной завесы
RunVlvDrench := BtnRunVlvDrench;

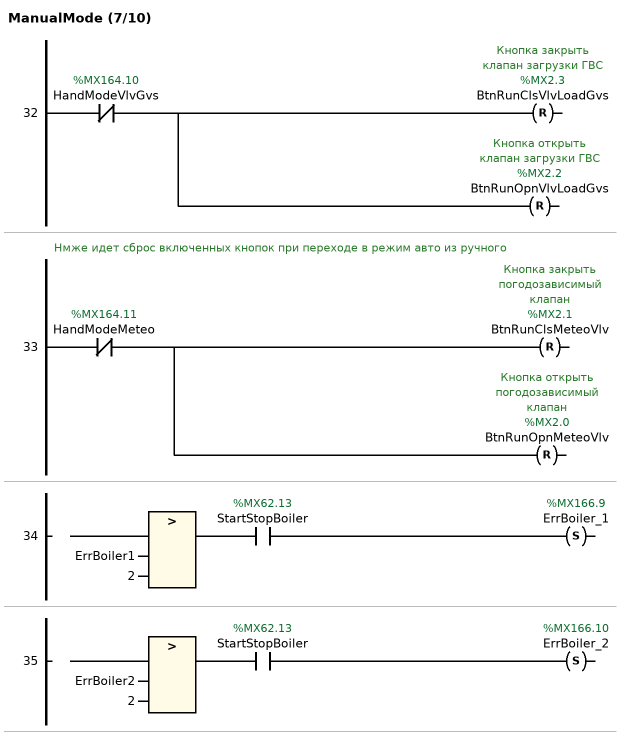
// NETWORK 32
//   HandModeVlvGvs: AT %MX164.10
//   BtnRunClsVlvLoadGvs: Кнопка закрыть клапан загрузки ГВС | AT %MX2.3
//   BtnRunOpnVlvLoadGvs: Кнопка открыть клапан загрузки ГВС | AT %MX2.2
_w6 := NOT HandModeVlvGvs;
BtnRunClsVlvLoadGvs R= _w6;
BtnRunOpnVlvLoadGvs R= _w6;

// NETWORK 33
// Нмже идет сброс включенных кнопок при переходе в режим авто из ручного
//   HandModeMeteo: AT %MX164.11
//   BtnRunClsMeteoVlv: Кнопка закрыть погодозависимый клапан | AT %MX2.1
//   BtnRunOpnMeteoVlv: Кнопка открыть погодозависимый клапан | AT %MX2.0
_w7 := NOT HandModeMeteo;
BtnRunClsMeteoVlv R= _w7;
BtnRunOpnMeteoVlv R= _w7;

// NETWORK 34
//   StartStopBoiler: AT %MX62.13
//   ErrBoiler_1: AT %MX166.9
ErrBoiler_1 S= ErrBoiler1 > 2 AND StartStopBoiler;

// NETWORK 35
//   StartStopBoiler: AT %MX62.13
//   ErrBoiler_2: AT %MX166.10
ErrBoiler_2 S= ErrBoiler2 > 2 AND StartStopBoiler;

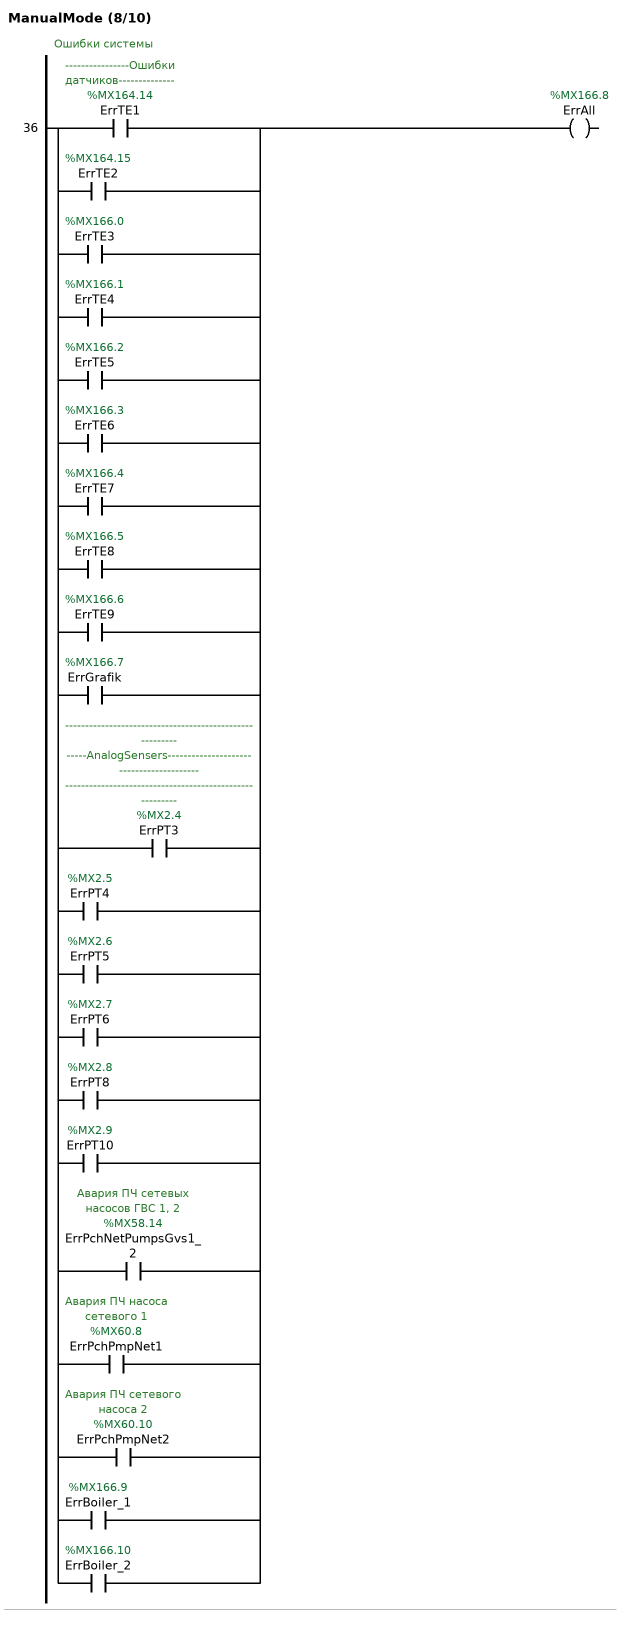
// NETWORK 36
// Ошибки системы
//   ErrTE1: ----------------Ошибки датчиков-------------- | AT %MX164.14
//   ErrTE2: AT %MX164.15
//   ErrTE3: AT %MX166.0
//   ErrTE4: AT %MX166.1
//   ErrTE5: AT %MX166.2
//   ErrTE6: AT %MX166.3
//   ErrTE7: AT %MX166.4
//   ErrTE8: AT %MX166.5
//   ErrTE9: AT %MX166.6
//   ErrGrafik: AT %MX166.7
//   ErrPT3: -------------------------------------------------------- -----AnalogSensers----------------------------------------- -------------------------------------------------------- | AT %MX2.4
//   ErrPT4: AT %MX2.5
//   ErrPT5: AT %MX2.6
//   ErrPT6: AT %MX2.7
//   ErrPT8: AT %MX2.8
//   ErrPT10: AT %MX2.9
//   ErrPchNetPumpsGvs1_2: Авария ПЧ сетевых насосов ГВС 1, 2 | AT %MX58.14
//   ErrPchPmpNet1: Авария ПЧ насоса сетевого 1 | AT %MX60.8
//   ErrPchPmpNet2: Авария ПЧ сетевого насоса 2 | AT %MX60.10
//   ErrBoiler_1: AT %MX166.9
//   ErrBoiler_2: AT %MX166.10
//   ErrAll: AT %MX166.8
ErrAll := ErrTE1 OR ErrTE2 OR ErrTE3 OR ErrTE4 OR ErrTE5 OR ErrTE6 OR ErrTE7 OR ErrTE8 OR ErrTE9 OR ErrGrafik OR ErrPT3 OR ErrPT4 OR ErrPT5 OR ErrPT6 OR ErrPT8 OR ErrPT10 OR ErrPchNetPumpsGvs1_2 OR ErrPchPmpNet1 OR ErrPchPmpNet2 OR ErrBoiler_1 OR ErrBoiler_2;

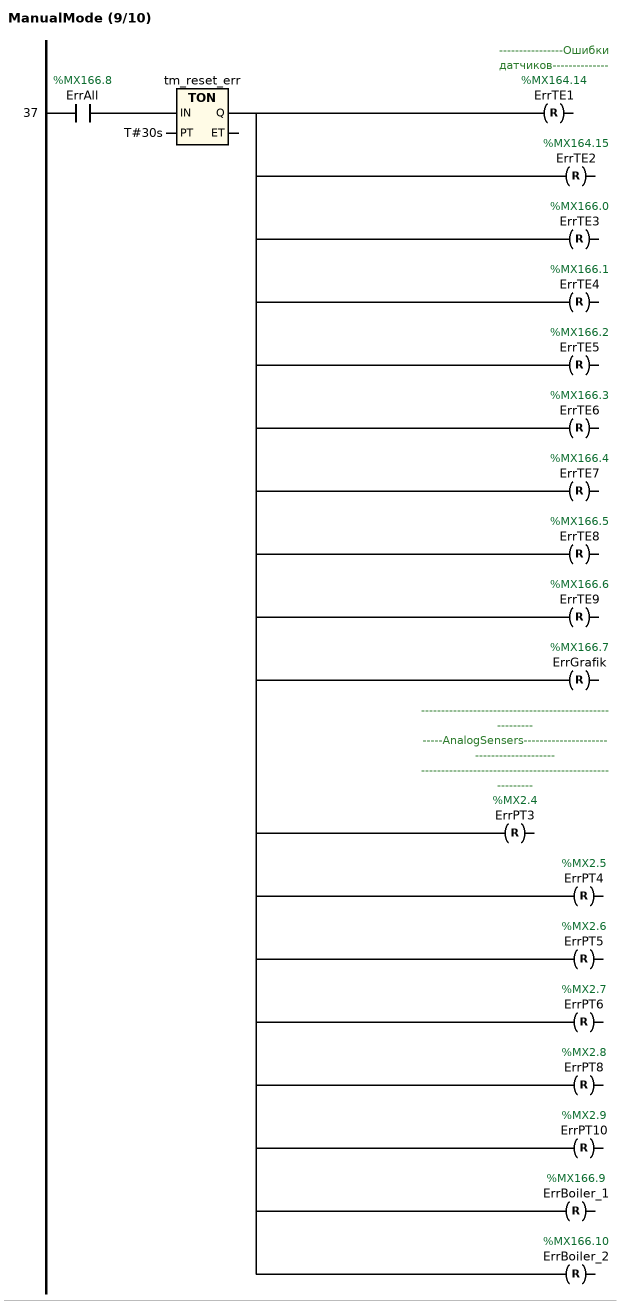
// NETWORK 37
//   ErrAll: AT %MX166.8
//   ErrTE1: ----------------Ошибки датчиков-------------- | AT %MX164.14
//   ErrTE2: AT %MX164.15
//   ErrTE3: AT %MX166.0
//   ErrTE4: AT %MX166.1
//   ErrTE5: AT %MX166.2
//   ErrTE6: AT %MX166.3
//   ErrTE7: AT %MX166.4
//   ErrTE8: AT %MX166.5
//   ErrTE9: AT %MX166.6
//   ErrGrafik: AT %MX166.7
//   ErrPT3: -------------------------------------------------------- -----AnalogSensers----------------------------------------- -------------------------------------------------------- | AT %MX2.4
//   ErrPT4: AT %MX2.5
//   ErrPT5: AT %MX2.6
//   ErrPT6: AT %MX2.7
//   ErrPT8: AT %MX2.8
//   ErrPT10: AT %MX2.9
//   ErrBoiler_1: AT %MX166.9
//   ErrBoiler_2: AT %MX166.10
tm_reset_err(IN := ErrAll, PT := T#30s); // TON
ErrTE1 R= tm_reset_err.Q;
ErrTE2 R= tm_reset_err.Q;
ErrTE3 R= tm_reset_err.Q;
ErrTE4 R= tm_reset_err.Q;
ErrTE5 R= tm_reset_err.Q;
ErrTE6 R= tm_reset_err.Q;
ErrTE7 R= tm_reset_err.Q;
ErrTE8 R= tm_reset_err.Q;
ErrTE9 R= tm_reset_err.Q;
ErrGrafik R= tm_reset_err.Q;
ErrPT3 R= tm_reset_err.Q;
ErrPT4 R= tm_reset_err.Q;
ErrPT5 R= tm_reset_err.Q;
ErrPT6 R= tm_reset_err.Q;
ErrPT8 R= tm_reset_err.Q;
ErrPT10 R= tm_reset_err.Q;
ErrBoiler_1 R= tm_reset_err.Q;
ErrBoiler_2 R= tm_reset_err.Q;

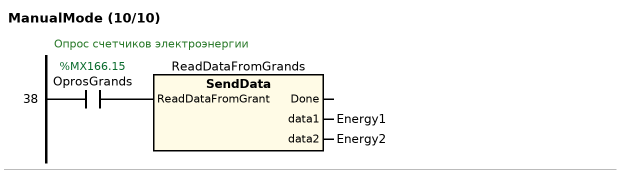
// NETWORK 38
// Опрос счетчиков электроэнергии
//   OprosGrands: AT %MX166.15
//   Energy1: AT %MD2000
//   Energy2: AT %MD2002
ReadDataFromGrands(ReadDataFromGrant := OprosGrands, data1 => Energy1, data2 => Energy2); // SendData

END_PROGRAM

// MyController/Application/SendData
FUNCTION_BLOCK SendData
VAR_INPUT
	ReadDataFromGrant: BOOL;
END_VAR
VAR_OUTPUT
	Done: BOOL;
	data1: DWORD;
	data2: DWORD;
END_VAR
VAR
	power1: SEND_RECV_MSG;
	ADDM_0: ADDM;
	SL1_adr: ADDRESS;
	Tx: ARRAY [1..10] OF BYTE:=[1,4,1,0,0,0,7,8];
	Rx: ARRAY [1..10] OF BYTE;
	
	power2: SEND_RECV_MSG;
	ADDM_1: ADDM;
	Tx2: ARRAY [1..10] OF BYTE:=[2,4,1,0,0,0,7,8];
	Rx2: ARRAY [1..10] OF BYTE;
	CRC2: WORD;
	tm_delay: TON;
	crc_1: CRC_16;
	crc_2: CRC_16;
	energy_1: array_to_float;
	energy_2: array_to_float;
END_VAR
VAR // added by the converter: edge detectors and wires of the graphical bodies
    _w1, _w2, _w3, _w4, _w5 : ANY;
END_VAR

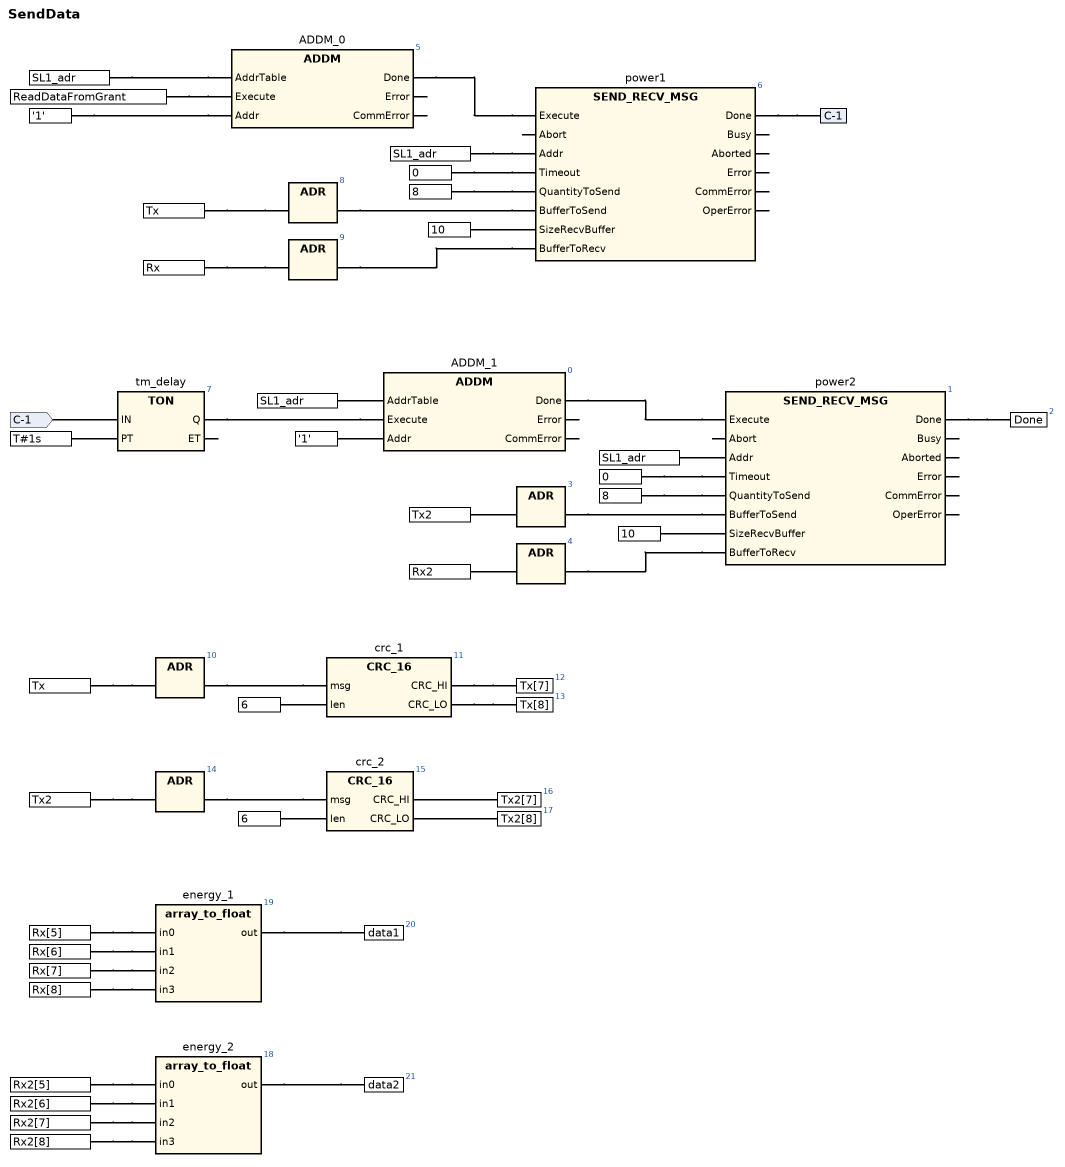
ADDM_1(AddrTable := SL1_adr, Execute := tm_delay.Q, Addr := '1'); // ADDM
power2(
    Execute := ADDM_1.Done,
    Addr := SL1_adr,
    Timeout := 0,
    QuantityToSend := 8,
    BufferToSend := _w1,
    SizeRecvBuffer := 10,
    BufferToRecv := _w2); // SEND_RECV_MSG
Done := power2.Done;
_w1 := ADR(Tx2);
_w2 := ADR(Rx2);
ADDM_0(AddrTable := SL1_adr, Execute := ReadDataFromGrant, Addr := '1'); // ADDM
power1(
    Execute := ADDM_0.Done,
    Addr := SL1_adr,
    Timeout := 0,
    QuantityToSend := 8,
    BufferToSend := _w3,
    SizeRecvBuffer := 10,
    BufferToRecv := _w4); // SEND_RECV_MSG
tm_delay(IN := _w5, PT := T#1s); // TON
_w3 := ADR(Tx);
_w4 := ADR(Rx);
crc_1(msg := ADR(Tx), len := 6); // CRC_16
Tx[7] := crc_1.CRC_HI;
Tx[8] := crc_1.CRC_LO;
crc_2(msg := ADR(Tx2), len := 6); // CRC_16
Tx2[7] := crc_2.CRC_HI;
Tx2[8] := crc_2.CRC_LO;
energy_2(in0 := Rx2[5], in1 := Rx2[6], in2 := Rx2[7], in3 := Rx2[8]); // array_to_float
energy_1(in0 := Rx[5], in1 := Rx[6], in2 := Rx[7], in3 := Rx[8]); // array_to_float
data1 := energy_1.out;
data2 := energy_2.out;

END_FUNCTION_BLOCK

// MyController/Application/CRC_16
FUNCTION_BLOCK CRC_16
VAR_INPUT
	msg: POINTER TO BYTE;//Сообщение
	len: WORD;// Длина сообщения для которого нужно посчитать CRC
END_VAR
VAR
tblCRChi: ARRAY[0..255] OF BYTE := 
[16#00, 16#C1, 16#81, 16#40, 16#01, 16#C0, 16#80, 16#41, 16#01, 16#C0, 16#80, 16#41, 16#00, 16#C1, 16#81,
16#40, 16#01, 16#C0, 16#80, 16#41, 16#00, 16#C1, 16#81, 16#40, 16#00, 16#C1, 16#81, 16#40, 16#01, 16#C0,
16#80, 16#41, 16#01, 16#C0, 16#80, 16#41, 16#00, 16#C1, 16#81, 16#40, 16#00, 16#C1, 16#81, 16#40, 16#01,
16#C0, 16#80, 16#41, 16#00, 16#C1, 16#81, 16#40, 16#01, 16#C0, 16#80, 16#41, 16#01, 16#C0, 16#80, 16#41,
16#00, 16#C1, 16#81, 16#40, 16#01, 16#C0, 16#80, 16#41, 16#00, 16#C1, 16#81, 16#40, 16#00, 16#C1, 16#81,
16#40, 16#01, 16#C0, 16#80, 16#41, 16#00, 16#C1, 16#81, 16#40, 16#01, 16#C0, 16#80, 16#41, 16#01, 16#C0,
16#80, 16#41, 16#00, 16#C1, 16#81, 16#40, 16#00, 16#C1, 16#81, 16#40, 16#01, 16#C0, 16#80, 16#41, 16#01,
16#C0, 16#80, 16#41, 16#00, 16#C1, 16#81, 16#40, 16#01, 16#C0, 16#80, 16#41, 16#00, 16#C1, 16#81, 16#40,
16#00, 16#C1, 16#81, 16#40, 16#01, 16#C0, 16#80, 16#41, 16#01, 16#C0, 16#80, 16#41, 16#00, 16#C1, 16#81,
16#40, 16#00, 16#C1, 16#81, 16#40, 16#01, 16#C0, 16#80, 16#41, 16#00, 16#C1, 16#81, 16#40, 16#01, 16#C0,
16#80, 16#41, 16#01, 16#C0, 16#80, 16#41, 16#00, 16#C1, 16#81, 16#40, 16#00, 16#C1, 16#81, 16#40, 16#01,
16#C0, 16#80, 16#41, 16#01, 16#C0, 16#80, 16#41, 16#00, 16#C1, 16#81, 16#40, 16#01, 16#C0, 16#80, 16#41,
16#00, 16#C1, 16#81, 16#40, 16#00, 16#C1, 16#81, 16#40, 16#01, 16#C0, 16#80, 16#41, 16#00, 16#C1, 16#81,
16#40, 16#01, 16#C0, 16#80, 16#41, 16#01, 16#C0, 16#80, 16#41, 16#00, 16#C1, 16#81, 16#40, 16#01, 16#C0,
16#80, 16#41, 16#00, 16#C1, 16#81, 16#40, 16#00, 16#C1, 16#81, 16#40, 16#01, 16#C0, 16#80, 16#41, 16#01,
16#C0, 16#80, 16#41, 16#00, 16#C1, 16#81, 16#40, 16#00, 16#C1, 16#81, 16#40, 16#01, 16#C0, 16#80, 16#41,
16#00, 16#C1, 16#81, 16#40, 16#01, 16#C0, 16#80, 16#41, 16#01, 16#C0, 16#80, 16#41, 16#00, 16#C1, 16#81,
16#40];

tblCRClo: ARRAY[0..255] OF BYTE := 
[16#00, 16#C0, 16#C1, 16#01, 16#C3, 16#03, 16#02, 16#C2, 16#C6, 16#06, 16#07, 16#C7, 16#05, 16#C5, 16#C4,
16#04, 16#CC, 16#0C, 16#0D, 16#CD, 16#0F, 16#CF, 16#CE, 16#0E, 16#0A, 16#CA, 16#CB, 16#0B, 16#C9, 16#09,
16#08, 16#C8, 16#D8, 16#18, 16#19, 16#D9, 16#1B, 16#DB, 16#DA, 16#1A, 16#1E, 16#DE, 16#DF, 16#1F, 16#DD,
16#1D, 16#1C, 16#DC, 16#14, 16#D4, 16#D5, 16#15, 16#D7, 16#17, 16#16, 16#D6, 16#D2, 16#12, 16#13, 16#D3,
16#11, 16#D1, 16#D0, 16#10, 16#F0, 16#30, 16#31, 16#F1, 16#33, 16#F3, 16#F2, 16#32, 16#36, 16#F6, 16#F7,
16#37, 16#F5, 16#35, 16#34, 16#F4, 16#3C, 16#FC, 16#FD, 16#3D, 16#FF, 16#3F, 16#3E, 16#FE, 16#FA, 16#3A,
16#3B, 16#FB, 16#39, 16#F9, 16#F8, 16#38, 16#28, 16#E8, 16#E9, 16#29, 16#EB, 16#2B, 16#2A, 16#EA, 16#EE,
16#2E, 16#2F, 16#EF, 16#2D, 16#ED, 16#EC, 16#2C, 16#E4, 16#24, 16#25, 16#E5, 16#27, 16#E7, 16#E6, 16#26,
16#22, 16#E2, 16#E3, 16#23, 16#E1, 16#21, 16#20, 16#E0, 16#A0, 16#60, 16#61, 16#A1, 16#63, 16#A3, 16#A2,
16#62, 16#66, 16#A6, 16#A7, 16#67, 16#A5, 16#65, 16#64, 16#A4, 16#6C, 16#AC, 16#AD, 16#6D, 16#AF, 16#6F,
16#6E, 16#AE, 16#AA, 16#6A, 16#6B, 16#AB, 16#69, 16#A9, 16#A8, 16#68, 16#78, 16#B8, 16#B9, 16#79, 16#BB,
16#7B, 16#7A, 16#BA, 16#BE, 16#7E, 16#7F, 16#BF, 16#7D, 16#BD, 16#BC, 16#7C, 16#B4, 16#74, 16#75, 16#B5,
16#77, 16#B7, 16#B6, 16#76, 16#72, 16#B2, 16#B3, 16#73, 16#B1, 16#71, 16#70, 16#B0, 16#50, 16#90, 16#91,
16#51, 16#93, 16#53, 16#52, 16#92, 16#96, 16#56, 16#57, 16#97, 16#55, 16#95, 16#94, 16#54, 16#9C, 16#5C,
16#5D, 16#9D, 16#5F, 16#9F, 16#9E, 16#5E, 16#5A, 16#9A, 16#9B, 16#5B, 16#99, 16#59, 16#58, 16#98, 16#88,
16#48, 16#49, 16#89, 16#4B, 16#8B, 16#8A, 16#4A, 16#4E, 16#8E, 16#8F, 16#4F, 16#8D, 16#4D, 16#4C, 16#8C,
16#44, 16#84, 16#85, 16#45, 16#87, 16#47, 16#46, 16#86, 16#82, 16#42, 16#43, 16#83, 16#41, 16#81, 16#80,
16#40];

Idx: WORD;
CRChi: BYTE;
CRClo: BYTE;
END_VAR
VAR_OUTPUT
	CRC_HI: BYTE;
	CRC_LO: BYTE;
END_VAR
VAR
END_VAR

CRChi:= 16#FF;
CRClo:= 16#FF;
WHILE len>0 DO
Idx := (CRChi XOR msg^) AND 16#FF;
CRChi := CRClo XOR tblCRChi[Idx];
CRClo := tblCRClo[idx];
len:=len-1;
msg:=msg+SIZEOF(msg^);
END_WHILE
CRC_HI:=CRChi;
CRC_LO:=CRClo;

END_FUNCTION_BLOCK

// MyController/Application/array_to_float
FUNCTION_BLOCK array_to_float
VAR_INPUT
	in0:BYTE;
	in1:BYTE;
	in2:BYTE;
	in3:BYTE;
END_VAR
VAR_OUTPUT
	out:DWORD;
END_VAR
VAR
	temp: DWORD;
END_VAR

temp:= in0;
out := SHL(temp,24);
temp:= in1;
out := out OR SHL(temp,16);
temp:= in2;
out := out OR SHL(temp,8);
temp:= in3;
out := out OR in3;

END_FUNCTION_BLOCK

// MyController/Application/year_month_day
PROGRAM year_month_day
VAR
	  uidResultRtcGet: UDINT;
      stGetDate: SysTimeRtc.RTS_SYSTIMEDATE; 
      uiGetMSecond: UINT; 
      uiGetYday: UINT; 
      uidResultConvertToDate: UDINT; 

	  
	  udiResultConvertToUtc: UDINT; 
      dwSetTimeStamp: DWORD;

      uidResultRtcSet: UDINT;
	  set_time: TON;
END_VAR
VAR // added by the converter: edge detectors and wires of the graphical bodies
    _s1 : RTS_SYSTIMEDATE;
    _w1, _w2, _w4 : ANY;
    _w3 : BOOL;
END_VAR

_w1 := SysTimeRtcGet(pResult := uidResultRtcGet);
// compose _s1 : RTS_SYSTIMEDATE
_s1.wYear := uiSetYear;
_s1.wMonth := uiSetMonth;
_s1.wDay := uiSetDay;
_s1.wHour := uiSetHour;
_s1.wMinute := uiSetMinute;
_s1.wSecond := uiSetSecond;
_s1.wMilliseconds := uiSetMSecond;
IF uidResultRtcGet = 16#0 THEN SysTimeRtcConvertUtcToDate(dwTimestampUtc := _w1, pDate := stGetDate); END_IF
_w2 := SysTimeRtcConvertDateToUtc(pDate := _s1, pdwTimestampUtc := dwSetTimeStamp);
udiResultConvertToUtc := _w2;
uiGetYear := stGetDate.RTS_SYSTIMEDATE;
uiGetMonth := stGetDate.wYear;
IF xCommandSetRtc AND _w3 THEN _w4 := SysTimeRtcSet(ulTimestamp := dwSetTimeStamp); END_IF
uiGetDay := stGetDate.wMonth;
uiGetHour := stGetDate.wDay;
uiGetMinute := stGetDate.wHour;
_w3 := udiResultConvertToUtc = 0;
uiGetSecond := stGetDate.wMinute;
uidResultRtcSet := _w4;
uiGetMSecond := stGetDate.wSecond;
uiGetDayOfWeek := stGetDate.wMilliseconds;
uiGetYday := stGetDate.wDayOfWeek;
set_time(IN := xCommandSetRtc, PT := T#1s); // TON
xCommandSetRtc R= set_time.Q;

END_PROGRAM

// MyController/Application/DQ
PROGRAM DQ
VAR
END_VAR

//------Модуль А1------------
Y0:=Rezerv;
Y1:=RunAlarm;
Y2:=RunSiren;
Y3:=RunPmpRcr1;
Y4:=RunPmpRcr2;
Y5:=RunPmpRcr3;
Y6:=RunPmpWtr1;
Y7:=RunPmpWtr2;
Y8:=RumPmpGvs1FromPch;
Y9:=RumPmpGvs2FromPch;
Y10:=StartPchGvs1_2;
Y11:=RunPmpNet1;//Y11:=RunPmpNet1FromNet;
Y12:=RunPmpNet2;//Y12:=RunPmpNet2FromNet;
Y13:=RunFan;
Y14:=RunPmpLoadGvs1;
Y15:=RunPmpLoadGvs2;

//------Модуль А1.1------------
_1Y0:=RunVlvDrench;
_1Y1:=RunOpnMeteoVlv;
_1Y2:=RunClsMeteoVlv;
_1Y3:=RunOpnVlvLoadGvs;
_1Y4:=RunClsVlvLoadGvs;

END_PROGRAM

// MyController/Application/CRC16
FUNCTION CRC16 : WORD
VAR_INPUT
	msg: POINTER TO BYTE;
	len: WORD;
END_VAR
VAR
tblCRChi: ARRAY[0..255] OF BYTE := 
[16#00, 16#C1, 16#81, 16#40, 16#01, 16#C0, 16#80, 16#41, 16#01, 16#C0, 16#80, 16#41, 16#00, 16#C1, 16#81,
16#40, 16#01, 16#C0, 16#80, 16#41, 16#00, 16#C1, 16#81, 16#40, 16#00, 16#C1, 16#81, 16#40, 16#01, 16#C0,
16#80, 16#41, 16#01, 16#C0, 16#80, 16#41, 16#00, 16#C1, 16#81, 16#40, 16#00, 16#C1, 16#81, 16#40, 16#01,
16#C0, 16#80, 16#41, 16#00, 16#C1, 16#81, 16#40, 16#01, 16#C0, 16#80, 16#41, 16#01, 16#C0, 16#80, 16#41,
16#00, 16#C1, 16#81, 16#40, 16#01, 16#C0, 16#80, 16#41, 16#00, 16#C1, 16#81, 16#40, 16#00, 16#C1, 16#81,
16#40, 16#01, 16#C0, 16#80, 16#41, 16#00, 16#C1, 16#81, 16#40, 16#01, 16#C0, 16#80, 16#41, 16#01, 16#C0,
16#80, 16#41, 16#00, 16#C1, 16#81, 16#40, 16#00, 16#C1, 16#81, 16#40, 16#01, 16#C0, 16#80, 16#41, 16#01,
16#C0, 16#80, 16#41, 16#00, 16#C1, 16#81, 16#40, 16#01, 16#C0, 16#80, 16#41, 16#00, 16#C1, 16#81, 16#40,
16#00, 16#C1, 16#81, 16#40, 16#01, 16#C0, 16#80, 16#41, 16#01, 16#C0, 16#80, 16#41, 16#00, 16#C1, 16#81,
16#40, 16#00, 16#C1, 16#81, 16#40, 16#01, 16#C0, 16#80, 16#41, 16#00, 16#C1, 16#81, 16#40, 16#01, 16#C0,
16#80, 16#41, 16#01, 16#C0, 16#80, 16#41, 16#00, 16#C1, 16#81, 16#40, 16#00, 16#C1, 16#81, 16#40, 16#01,
16#C0, 16#80, 16#41, 16#01, 16#C0, 16#80, 16#41, 16#00, 16#C1, 16#81, 16#40, 16#01, 16#C0, 16#80, 16#41,
16#00, 16#C1, 16#81, 16#40, 16#00, 16#C1, 16#81, 16#40, 16#01, 16#C0, 16#80, 16#41, 16#00, 16#C1, 16#81,
16#40, 16#01, 16#C0, 16#80, 16#41, 16#01, 16#C0, 16#80, 16#41, 16#00, 16#C1, 16#81, 16#40, 16#01, 16#C0,
16#80, 16#41, 16#00, 16#C1, 16#81, 16#40, 16#00, 16#C1, 16#81, 16#40, 16#01, 16#C0, 16#80, 16#41, 16#01,
16#C0, 16#80, 16#41, 16#00, 16#C1, 16#81, 16#40, 16#00, 16#C1, 16#81, 16#40, 16#01, 16#C0, 16#80, 16#41,
16#00, 16#C1, 16#81, 16#40, 16#01, 16#C0, 16#80, 16#41, 16#01, 16#C0, 16#80, 16#41, 16#00, 16#C1, 16#81,
16#40];

tblCRClo: ARRAY[0..255] OF BYTE := 
[16#00, 16#C0, 16#C1, 16#01, 16#C3, 16#03, 16#02, 16#C2, 16#C6, 16#06, 16#07, 16#C7, 16#05, 16#C5, 16#C4,
16#04, 16#CC, 16#0C, 16#0D, 16#CD, 16#0F, 16#CF, 16#CE, 16#0E, 16#0A, 16#CA, 16#CB, 16#0B, 16#C9, 16#09,
16#08, 16#C8, 16#D8, 16#18, 16#19, 16#D9, 16#1B, 16#DB, 16#DA, 16#1A, 16#1E, 16#DE, 16#DF, 16#1F, 16#DD,
16#1D, 16#1C, 16#DC, 16#14, 16#D4, 16#D5, 16#15, 16#D7, 16#17, 16#16, 16#D6, 16#D2, 16#12, 16#13, 16#D3,
16#11, 16#D1, 16#D0, 16#10, 16#F0, 16#30, 16#31, 16#F1, 16#33, 16#F3, 16#F2, 16#32, 16#36, 16#F6, 16#F7,
16#37, 16#F5, 16#35, 16#34, 16#F4, 16#3C, 16#FC, 16#FD, 16#3D, 16#FF, 16#3F, 16#3E, 16#FE, 16#FA, 16#3A,
16#3B, 16#FB, 16#39, 16#F9, 16#F8, 16#38, 16#28, 16#E8, 16#E9, 16#29, 16#EB, 16#2B, 16#2A, 16#EA, 16#EE,
16#2E, 16#2F, 16#EF, 16#2D, 16#ED, 16#EC, 16#2C, 16#E4, 16#24, 16#25, 16#E5, 16#27, 16#E7, 16#E6, 16#26,
16#22, 16#E2, 16#E3, 16#23, 16#E1, 16#21, 16#20, 16#E0, 16#A0, 16#60, 16#61, 16#A1, 16#63, 16#A3, 16#A2,
16#62, 16#66, 16#A6, 16#A7, 16#67, 16#A5, 16#65, 16#64, 16#A4, 16#6C, 16#AC, 16#AD, 16#6D, 16#AF, 16#6F,
16#6E, 16#AE, 16#AA, 16#6A, 16#6B, 16#AB, 16#69, 16#A9, 16#A8, 16#68, 16#78, 16#B8, 16#B9, 16#79, 16#BB,
16#7B, 16#7A, 16#BA, 16#BE, 16#7E, 16#7F, 16#BF, 16#7D, 16#BD, 16#BC, 16#7C, 16#B4, 16#74, 16#75, 16#B5,
16#77, 16#B7, 16#B6, 16#76, 16#72, 16#B2, 16#B3, 16#73, 16#B1, 16#71, 16#70, 16#B0, 16#50, 16#90, 16#91,
16#51, 16#93, 16#53, 16#52, 16#92, 16#96, 16#56, 16#57, 16#97, 16#55, 16#95, 16#94, 16#54, 16#9C, 16#5C,
16#5D, 16#9D, 16#5F, 16#9F, 16#9E, 16#5E, 16#5A, 16#9A, 16#9B, 16#5B, 16#99, 16#59, 16#58, 16#98, 16#88,
16#48, 16#49, 16#89, 16#4B, 16#8B, 16#8A, 16#4A, 16#4E, 16#8E, 16#8F, 16#4F, 16#8D, 16#4D, 16#4C, 16#8C,
16#44, 16#84, 16#85, 16#45, 16#87, 16#47, 16#46, 16#86, 16#82, 16#42, 16#43, 16#83, 16#41, 16#81, 16#80,
16#40];

Idx: WORD;
CRChi: BYTE := 16#FF;
CRClo: BYTE := 16#FF;
i: INT := 0;
END_VAR

WHILE len>=0 DO
Idx := (CRChi XOR msg^) AND 16#FF;
CRChi := CRClo XOR tblCRChi[Idx];
CRClo := tblCRClo[idx];
len:=len-1;
msg:=msg+1;
END_WHILE
CRC16:=(SHL(CRChi,8)) OR CRClo;

END_FUNCTION
